# B&R Automation Studio project AriesV2
Automation Studio 4.2.4.149

## Configuration Config_3500HS

### Task classes (Cpu.sw)
```
Cyclic#1:
  runFirst <- Libraries.wbrServices.InitSP.runFirst.prg (BuildOptions=-D "str(x)=#x" -D AS_PROJ=str($(AS_PROJECT_NAME)) -D AS_CFG=str($(AS_CONFIGURATION)) -D "AS_VERS=str($(AS_VERSION))" -D "AS_USER=str($(AS_USER_NAME))" -D "AS_CMPNY=str($(AS_COMPANY_NAME))")
  ForceIO1 <- HMI.ForceIO.prg
  ForceIO <- HMI.ForceIO.prg
Cyclic#8:
  wbrService <- Libraries.wbrServices.Cyclic.wbrService.prg
  HMITableMa <- HMI.HMITableManager.prg
  Recipe_Han <- Auxiliary_Services_Control.Recipe_Handling.prg  // Call functions that manage structures pertaining to params
  hmilogic <- HMI.hmilogic.prg
  ComLogger <- Auxiliary_Services_Control.ComLogger.prg [disabled]
  File_Handl <- Auxiliary_Services_Control.File_Handling.prg
DataObjects: ethIPcon
VcDataObjects: VisuW1 <- HMI.VisuW1.dob
Binaries: TCData, vccpwd, vccbtn, vcpdvnc, arialbd, vcmgr, vctcal, vcfile, vccnum, vcfntttf, vcgclass, vcbclass, vccshape, vccstr, vccalarm, vccscale, arial, vcalarm, vcdsloc, vcchtml, vccdt, vccbmp, vcshared, vcxml, vccurl, vcrt, vcctext, vcnet, vcclbox, vcdsint, vcpdsw, vccovl, vccline, VisuW101, VisuW102, VisuW103, vera, vccgauge, vcpfx20, TC, Data_Log, MAPP_Alm, MAPP_Rec, MAPP_Web, MAPP_File, MAPP_Cfg, iomap, asfw, sysconf, ashwd, arconfig, Alarm, vcctrend, vccpopup, vccddbox, vccpiech, vcpkat, verabd, Visu, Visu02, Visu03, Visu01, Axes, Config_1, MAPP_Com, Recipe, File_Mgmt, vccslider, Acp10Map1, User, Role, Data, Config, VisuW03, VisuW02, VisuW01, acp10cfg, Acp10map, Acp10sys, vcpfar00
Libraries: wbrsprintf, FileIO, AsXml, standard, runtime, astime, brsystem, sys_lib, AsANSL, AsARCfg, AsBrMath, AsBrStr, DataObj, AsTCP, AsUDP, AsUSB, MpCom, MpAlarm, MpFile, MpRecipe, MpWebXs, AsArSdm, AsIecCon, operator, AsIOTime, AsMem, AsArLog, AsArProf, MTBasics, MTTypes, MTFilter, jgLibC, MTData, ArTextSys, AsICMP, bglibasWBR, MAPPSuppor, wbrFltUtil, wbrListSvc, wbrLogSvc, wbrMemSvc, wbrPingSvc, vcresman, arsvcreg, ashw, AsMbTCP, AsSafety, powerlnk
```

### MAPP_Cfg.mprecipecsv - X20CP1301/mapp/MAPP_Cfg.mprecipecsv
```
Element Config_CSV_MpLink (Type=mprecipecsv)
  mapp.Recipe.Csv:
    Format:
      DecimalMark = .
```

## Configuration Config_Deployment

### Task classes (Cpu.sw)
```
Cyclic#1 (cycle 4000 us, tolerance 0 us):
  ForceIO <- HMI.ForceIO.prg
  Creaser <- Application.Creaser.prg
  ForceIO1 <- HMI.ForceIO.prg
Cyclic#8 (cycle 8000 us, tolerance 30000000 us):
  LineContro <- MotionControl.LineControl.prg
  Recipe_Han <- Auxiliary_Services_Control.Recipe_Handling.prg
  hmilogic <- HMI.hmilogic.prg
  HMITableMa <- HMI.HMITableManager.prg
  File_Handl <- Auxiliary_Services_Control.File_Handling.prg
  ComLogger <- Auxiliary_Services_Control.ComLogger.prg
DataObjects: ethIPcon
NcDataObjects: acp10etxen <- acp10etxen.dob, Axisa <- Axisobj.Axisa.dob, Axisi <- Axisobj.Axisi.dob
VcDataObjects: Visu1 <- HMI.Visu.dob
Binaries: vccpwd, vccbtn, arialbd, vcfile, vccnum, vcfntttf, vcgclass, vcbclass, vccshape, vccstr, vccalarm, vccscale, arial, vcalarm, vcdsloc, vcchtml, vccdt, vccbmp, vcshared, vcxml, vccurl, vcrt, vcctext, vcclbox, vcdsint, vcpdsw, vccovl, vccline, vera, vcpfar00, vcpkat, vccddbox, vccpopup, vcnet, vctcal, vcmgr, vcpdvnc, udbdef, Acp10sys, TCData, Visu102, Visu101, Visu103, Alarm, ashwd, asfw, MAPP_Cfg, MAPP_File, MAPP_Web, MAPP_Rec, MAPP_Alm, Data_Log, arconfig, sysconf, iomap, Config, acp10cfg, Acp10map, VisuW101, vcpfx20, vcctrend, vccpiech, verabd, Visu, Visu02, Visu03, Visu01, Axes, Config_1, MAPP_Com, Recipe, File_Mgmt, vccslider, Acp10Map1, User, Role, Data, VisuW03, VisuW02, VisuW01, TC, vccgauge, VisuW103, VisuW102
Libraries: FileIO, AsXml, standard, runtime, astime, brsystem, sys_lib, AsANSL, AsARCfg, AsBrMath, AsBrStr, DataObj, AsTCP, AsUDP, AsUSB, AsArSdm, AsIecCon, operator, AsIOTime, AsMem, AsArLog, AsArProf, AsICMP, Acp10man, Acp10par, NcGlobal, Acp10_MC, MpAxis, MpCom, wbrsprintf, wbrPingSvc, wbrMemSvc, wbrLogSvc, wbrListSvc, wbrFltUtil, MpWebXs, MpRecipe, MpFile, MpAlarm, MAPPSuppor, jgLibC, bglibasWBR, vcresman, arsvcreg, powerlnk, Acp10sim, ashw, AsMbTCP, AsSafety, ArTextSys
```

### Hardware
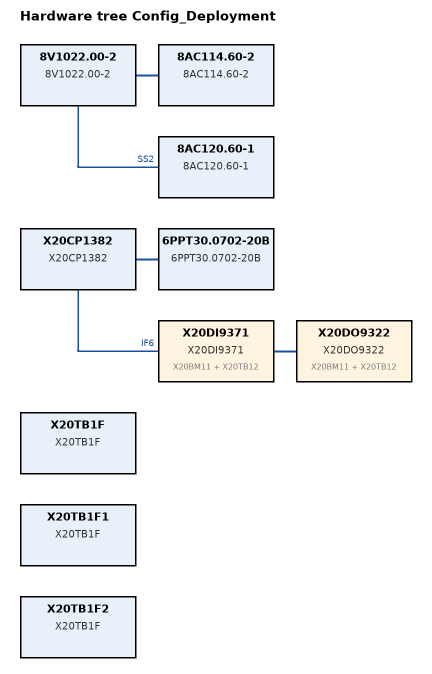
```
6PPT30.0702-20B : 6PPT30.0702-20B v1.1.0.0  [ETH1 -> X20CP1382.IF2 (NodeNumber=1)]
  Terminal = true
  Startmode = 1
  ShowBootlogoVNC = 1
  Mode = Manual
  InternetAddress = 192.168.10.20
  DefaultGateway = 192.168.10.1
  Subnetmask = 255.255.255.0
  Displaybrightness = 75
  SelectedFavoriteVNC = 192.168.10.10
  Favorites_VNC1 = 192.168.10.10
  PasswordVNC = 
  PasswordCIFS = 
  PasswordService = 
  PPTImage = PPT_30_V1.1.1
  VncRefreshRate = 200
8AC114.60-2 : 8AC114.60-2 v1.0.0.8  [SS -> 8V1022.00-2.SS1; PLK1 -> X20CP1382.IF3 (NodeNumber=2)]
8AC120.60-1 : 8AC120.60-1 v1.0.0.2  [SS -> 8V1022.00-2.SS2]
8V1022.00-2 : 8V1022.00-2 v1.0.0.2
  AxisIsPeriodic_r1 = on
  BothEndSwitchesAreNormallyOpen_r1 = on
  QuickStopIsNormallyOpen_r1 = on
X20BM11 : X20BM11 v1.0.0.1  [X2X1 -> X20CP1382.IF6]
X20BM11a : X20BM11 v1.0.0.1  [X2X1 -> X20BM11.X2X2]
X20CP1382 : X20CP1382 v1.3.0.0  [X1 -> X1.SL; X2 -> X2.SL; X3 -> X3.SL]
  Module X1 (Type=X1, Virtual=true, Version=1.0.0.0)
    Connection (Connector=SS1, TargetModule=X20TB1F, TargetConnector=SS)
    Connection (Connector=SL, TargetModule=X20CP1382, TargetConnector=X1)
  Module X2 (Type=X2, Virtual=true, Version=1.0.0.0)
    Connection (Connector=SS1, TargetModule=X20TB1F1, TargetConnector=SS)
    Connection (Connector=SL, TargetModule=X20CP1382, TargetConnector=X2)
  Module X3 (Type=X3, Virtual=true, Version=1.0.0.0)
    Connection (Connector=SS1, TargetModule=X20TB1F2, TargetConnector=SS)
    Connection (Connector=SL, TargetModule=X20CP1382, TargetConnector=X3)
  Connector IF2:
    ActivateDevice = 1
    HostName = x20cpu
    Mode = Manual
    InternetAddress = 192.168.10.10
    SubnetMask = 255.255.255.0
    InaNodeNumber = 0
    Vnc1
    VncVcObjectName1 = Visup
    VncKeyMappingFile1 = VC\PS2-Keyboard4.dis
    VncRefreshRate1 = 200
  Connector IF3:
    CycleTime = 4000
  Connector IF6:
    CycleTime = 4000
  ConfigurationID = AriesV2_Config_Test
  UserPartitionSize = 256
  UserRamSize = 5000
  RemMemSize = 25000
  PermanentPvSize = 15000
  VolatileGlobalPvSize = 300000
  RebootReset = 2
  RebootPowerfail = 2
  TimerDeviceType = EPLX2X
  TimerDevice = X20CP1382.IF3
  TaskClassIdleTime = 8000
  Cyclic1Duration = 4000
  Cyclic1Tolerance = 0
  Cyclic2Duration = 16000
  Cyclic2Tolerance = 16000
  Cyclic3Duration = 48000
  Cyclic3Tolerance = 48000
  Cyclic4Duration = 96000
  Cyclic4Tolerance = 96000
  Cyclic5Duration = 200000
  Cyclic5Tolerance = 200000
  Cyclic6Duration = 496000
  Cyclic6Tolerance = 496000
  Cyclic7Duration = 1000000
  Cyclic7Tolerance = 1000000
  Cyclic8Duration = 8000
  Cyclic8Tolerance = 30000000
  FileDevice1
  FileDeviceName1 = ROOT
  FileDevicePath1 = F:\
  FileDevice2
  FileDeviceName2 = Config
  FileDevicePath2 = F:\Config
  FileDevice3
  FileDeviceName3 = Recipe
  FileDevicePath3 = F:\Recipe
  FileDevice4
  FileDeviceName4 = Process
  FileDevicePath4 = F:\Process
  FtpUser1
  FtpUsername1 = admin
  FtpUserPassword1 = tXcQUdKIsoY/H/jtKSqzHLRzyWbO/eZFb+QmJVs8vuM=
  FtpUserSalt1 = fFlgpUU6
  FTPAccessRight1 = 0
  FTPdevice1 = ALL
  FtpUser2
  FtpUsername2 = user
  FtpUserPassword2 = M/sBBWLbPcMSL0ECBo9+NNWk5QFExAfaSSh+paOlJpQ=
  FtpUserSalt2 = diDYFxUT
  FTPAccessRight2 = 0
  FTPMSpath2 = /
X20DI9371 : X20DI9371 v1.0.1.3  [SS1 -> X20TB12.SS; SL -> X20BM11.SL1]
  Supervision = off
X20DO9322 : X20DO9322 v1.0.3.0  [SS1 -> X20TB12a.SS; SL -> X20BM11a.SL1]
  Supervision = off
X20TB12 : X20TB12 v1.0.0.0
X20TB12a : X20TB12 v1.0.0.0
X20TB1F : X20TB1F v1.0.0.0
X20TB1F1 : X20TB1F v1.0.0.0
X20TB1F2 : X20TB1F v1.0.0.0
```

### Acp10cfg.ncc - X20CP1382/Motion/Acp10cfg.ncc
```
NcConfiguration (Version=3.16.1, NcSwId=Acp10)
  ACP10CF1_typ:
    cnt_nettrc_rec_drive = 1500
    bufsize_trace_upload = 1200
    tc_nc_man_task = Cyclic #1
    glob_pv_as_ncobject = Yes
    ncsys_dl_broadcast = Yes
    ncsys_dl_acp_reset = Yes
    safemc_log_err_to_ax = Yes
    network_init:
      ncsw_init_execute = Yes
      automatic_execute = Yes
      node_nr_warning = Yes
      net_err_before_ncact = Yes
    nettrc:
      enter_parsecrec = Yes
      enter_ncaction = Yes
      save_ring_startidx = Yes
    cam_prof_download:
      cam_dat_dl_parallel = No
      tc_cam_dl_parallel = Task class for NC Manager task
    plk_if[0]:
      if_name = IF3
      tc_CycDat_PLCopen = Task class for NC Manager task
      mc_broadcast_extdat = No
```

### MAPP_File.mpfilemanagerui - X20CP1382/mapp/MAPP_File.mpfilemanagerui
```
Element File_Manager_MpLink (Type=mpfilemanagerui)
```

## Configuration Config_Test

CPU X20CP1584, AutomationRuntime B4.26, Build 4.1.2, Vc V4.26.3, Safety 0.0

CPU X20CP1585, AutomationRuntime B4.26, Build 4.1.2, Vc V4.26.3, Safety 1.5

### Task classes (Cpu.sw)
```
Cyclic#1 (cycle 8000 us, tolerance 0 us):
  ForceIO <- HMI.ForceIO.prg
  Creaser <- Application.Creaser.prg
  ForceIO1 <- HMI.ForceIO.prg
Cyclic#8 (cycle 8000 us, tolerance 30000000 us):
  LineContro <- MotionControl.LineControl.prg
  Recipe_Han <- Auxiliary_Services_Control.Recipe_Handling.prg
  hmilogic <- HMI.hmilogic.prg
  HMITableMa <- HMI.HMITableManager.prg
  File_Handl <- Auxiliary_Services_Control.File_Handling.prg
  ComLogger <- Auxiliary_Services_Control.ComLogger.prg
DataObjects: ethIPcon
NcDataObjects: acp10etxen <- acp10etxen.dob, Axisa <- Axisobj.Axisa.dob, Axisi <- Axisobj.Axisi.dob
VcDataObjects: Visu1 <- HMI.Visu.dob
Binaries: vccpwd, vccbtn, arialbd, vcfile, vccnum, vcfntttf, vcgclass, vcbclass, vccshape, vccstr, vccalarm, vccscale, arial, vcalarm, vcdsloc, vcchtml, vccdt, vccbmp, vcshared, vcxml, vccurl, vcrt, vcctext, vcclbox, vcdsint, vcpdsw, vccovl, vccline, VisuW102, VisuW103, vera, vccgauge, TC, vcpfar00, VisuW01, VisuW02, VisuW03, Data, Role, User, Acp10Map1, vccslider, File_Mgmt, Recipe, MAPP_Com, Config_1, Axes, Visu01, Visu03, Visu02, Visu, verabd, vcpkat, vccpiech, vccddbox, vccpopup, vcctrend, vcpfx20, VisuW101, vcnet, vctcal, vcmgr, vcpdvnc, Acp10map, acp10cfg, Config, iomap, sysconf, arconfig, Data_Log, MAPP_Alm, MAPP_Rec, MAPP_Web, MAPP_File, MAPP_Cfg, asfw, ashwd, Alarm, udbdef, Acp10sys, TCData
Libraries: FileIO, AsXml, standard, runtime, astime, brsystem, sys_lib, AsANSL, AsARCfg, AsBrMath, AsBrStr, DataObj, AsTCP, AsUDP, AsUSB, AsArSdm, AsIecCon, operator, AsIOTime, AsMem, AsArLog, AsArProf, AsICMP, Acp10man, Acp10par, NcGlobal, Acp10_MC, MpAxis, MpCom, wbrsprintf, wbrPingSvc, wbrMemSvc, wbrLogSvc, wbrListSvc, wbrFltUtil, MpWebXs, MpRecipe, MpFile, MpAlarm, MAPPSuppor, jgLibC, bglibasWBR, vcresman, AsSafety, AsMbTCP, ashw, arsvcreg, powerlnk, Acp10sim
```

### Task classes (Cpu.sw)
```
Cyclic#1 (cycle 8000 us, tolerance 0 us):
  ForceIO <- HMI.ForceIO.prg
  Creaser <- Application.Creaser.prg
  ForceIO1 <- HMI.ForceIO.prg
DataObjects: ethIPcon
NcDataObjects: acp10etxen <- acp10etxen.dob, Axisa <- Axisobj.Axisa.dob, Axisi <- Axisobj.Axisi.dob
Binaries: TCData, Acp10sys, udbdef, Acp10map, acp10cfg, Config, iomap, sysconf, arconfig, Data_Log, MAPP_Alm, MAPP_Rec, MAPP_Web, MAPP_File, MAPP_Cfg, asfw, ashwd, Alarm, vccpwd, vccbtn, arialbd, vcfile, vccnum, vcfntttf, vcgclass, vcbclass, vccshape, vccstr, vccalarm, vccscale, arial, vcalarm, vcdsloc, vcchtml, vccdt, vccbmp, vcshared, vcxml, vccurl, vcrt, vcctext, vcclbox, vcdsint, vcpdsw, vccovl, vccline, VisuW102, VisuW103, vera, vccgauge, TC, vcpfar00, VisuW01, VisuW02, VisuW03, Data, Role, User, Acp10Map1, vccslider, File_Mgmt, Recipe, MAPP_Com, Config_1, Axes, Visu01, Visu03, Visu02, Visu, verabd, vcpkat, vccpiech, vccddbox, vccpopup, vcctrend, vcpfx20, VisuW101, vcnet, vctcal, vcmgr, vcpdvnc
Libraries: FileIO, AsXml, standard, runtime, astime, brsystem, sys_lib, AsANSL, AsARCfg, AsBrMath, AsBrStr, DataObj, AsTCP, AsUDP, AsUSB, AsArSdm, AsIecCon, operator, AsIOTime, AsMem, AsArLog, AsArProf, AsICMP, powerlnk, Acp10man, Acp10par, NcGlobal, Acp10_MC, MTBasics, MTTypes, MpAxis, MpCom, wbrsprintf, wbrPingSvc, wbrMemSvc, wbrLogSvc, wbrListSvc, wbrFltUtil, MTProfile, MTFilter, MTData, MpWebXs, MpRecipe, MpFile, MpAlarm, MAPPSuppor, jgLibC, bglibasWBR, ArTextSys, vcresman, AsSafety, AsMbTCP, ashw, arsvcreg
```

### Task classes (Cpu.sw)
```
Cyclic#1 (cycle 8000 us, tolerance 0 us):
  runFirst <- Libraries.wbrServices.InitSP.runFirst.prg (BuildOptions=-D "str(x)=#x" -D AS_PROJ=str($(AS_PROJECT_NAME)) -D AS_CFG=str($(AS_CONFIGURATION)) -D "AS_VERS=str($(AS_VERSION))" -D "AS_USER=str($(AS_USER_NAME))" -D "AS_CMPNY=str($(AS_COMPANY_NAME))")
  ForceIO1 <- HMI.ForceIO.prg
  ForceIO <- HMI.ForceIO.prg
Cyclic#8 (cycle 8000 us, tolerance 30000000 us):
  wbrService <- Libraries.wbrServices.Cyclic.wbrService.prg
  HMITableMa <- HMI.HMITableManager.prg
  Recipe_Han <- Auxiliary_Services_Control.Recipe_Handling.prg  // Call functions that manage structures pertaining to params
  hmilogic <- HMI.hmilogic.prg
  ComLogger <- Auxiliary_Services_Control.ComLogger.prg
  File_Handl <- Auxiliary_Services_Control.File_Handling.prg
DataObjects: ethIPcon
Binaries: vccpwd, vccbtn, arialbd, vcfile, vccnum, vcfntttf, vcgclass, vcbclass, vccshape, vccstr, vccalarm, vccscale, arial, vcalarm, vcdsloc, vcchtml, vccdt, vccbmp, vcshared, vcxml, vccurl, vcrt, vcctext, vcclbox, vcdsint, vcpdsw, vccovl, vccline, VisuW102, VisuW103, vera, vccgauge, Alarm, ashwd, asfw, MAPP_Cfg, MAPP_File, MAPP_Web, MAPP_Rec, MAPP_Alm, Data_Log, TC, vcpfar00, Acp10sys, Acp10map, acp10cfg, VisuW01, VisuW02, VisuW03, Config, Data, Role, User, Acp10Map1, vccslider, File_Mgmt, Recipe, MAPP_Com, Config_1, Axes, Visu01, Visu03, Visu02, Visu, verabd, vcpkat, vccpiech, vccddbox, vccpopup, vcctrend, arconfig, sysconf, iomap, vcpfx20, VisuW101, vcnet, vctcal, vcmgr, vcpdvnc, TCData
Libraries: wbrsprintf, FileIO, AsXml, standard, runtime, astime, brsystem, sys_lib, AsANSL, AsARCfg, AsBrMath, AsBrStr, DataObj, AsTCP, AsUDP, AsUSB, MpCom, MpAlarm, MpFile, MpRecipe, MpWebXs, AsArSdm, AsIecCon, operator, AsIOTime, AsMem, AsArLog, AsArProf, MTBasics, MTTypes, MTFilter, jgLibC, MTData, ArTextSys, AsICMP, bglibasWBR, MAPPSuppor, wbrFltUtil, wbrListSvc, wbrLogSvc, wbrMemSvc, wbrPingSvc, vcresman, arsvcreg, powerlnk, AsSafety, AsMbTCP, ashw
```

### Hardware
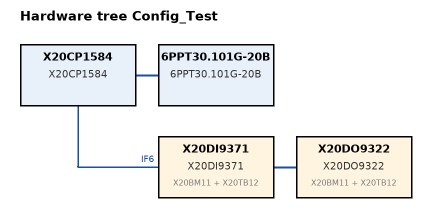
```
6PPT30.101G-20B : 6PPT30.101G-20B v1.1.0.0  [ETH1 -> X20CP1584.IF2 (NodeNumber=1)]
  Terminal = true
  PasswordVNC = 
  PasswordCIFS = 
  PasswordService = 
  VncKeyMappingFile = VC\6PPT30.101G-20B.dis
  VncPortNumber = 5901
X20BM11 : X20BM11 v1.0.0.1  [X2X1 -> X20CP1584.IF6]
X20BM11a : X20BM11 v1.0.0.1  [X2X1 -> X20BM11.X2X2]
X20CP1584 : X20CP1584 v1.3.2.0
  Connector IF2:
    ActivateDevice = 1
    EthInterfaceRedundant = 0
    HostName = x20cpu
    Mode = Manual
    InternetAddress = 192.168.10.10
    SubnetMask = 255.255.255.0
    Vnc1
    VncVcObjectName1 = Visu1
    VncKeyMappingFile1 = VC\PS2-Keyboard4.dis
    VncRefreshRate1 = 200
  Connector IF3:
    EplInterfaceRedundant = 0
    CycleTime = 8000
    EplEthInterfaceRedundant = 0
  Connector IF6:
    CycleTime = 8000
  ConfigurationID = AriesV2_Config_Test
  UserRamSize = 5000
  RemMemSize = 25000
  PermanentPvSize = 15000
  VolatileGlobalPvSize = 300000
  RebootReset = 2
  RebootPowerfail = 2
  TimerDeviceType = EPLX2X
  TimerDevice = X20CP1584.IF3
  TaskClassIdleTime = 8000
  Cyclic1Duration = 8000
  Cyclic1Tolerance = 0
  Cyclic2Duration = 16000
  Cyclic2Tolerance = 16000
  Cyclic3Duration = 48000
  Cyclic3Tolerance = 48000
  Cyclic4Duration = 96000
  Cyclic4Tolerance = 96000
  Cyclic5Duration = 200000
  Cyclic5Tolerance = 200000
  Cyclic6Duration = 496000
  Cyclic6Tolerance = 496000
  Cyclic7Duration = 1000000
  Cyclic7Tolerance = 1000000
  Cyclic8Duration = 8000
  Cyclic8Tolerance = 30000000
  FileDevice1
  FileDeviceName1 = ROOT
  FileDevicePath1 = F:\
  FileDevice2
  FileDeviceName2 = Config
  FileDevicePath2 = F:\Config
  FileDevice3
  FileDeviceName3 = Recipe
  FileDevicePath3 = F:\Recipe
  FileDevice4
  FileDeviceName4 = Process
  FileDevicePath4 = F:\Process
X20DI9371 : X20DI9371 v1.0.2.0  [SS1 -> X20TB12.SS; SL -> X20BM11.SL1]
  Supervision = off
X20DO9322 : X20DO9322 v1.0.3.0  [SS1 -> X20TB12a.SS; SL -> X20BM11a.SL1]
  Supervision = off
X20TB12 : X20TB12 v1.0.0.0
X20TB12a : X20TB12 v1.0.0.0
```

### Acp10map.ncm - X20CP1382/Motion/Acp10map.ncm
```
NcMapping (NcSwId=Acp10, DisabledNodesAreHidden=False)
  NcObject Axis1 (ModuleId=8V1022.00-2, Type=ncAXIS, Channel=1, AcoposSimulation=Complete, InitParameter=Axisi, AcoposParameter=Axisa, AdditionalData=PLCopen_ModPos="1000,1" , Disabled=FALSE, ModuleDisabled=FALSE)
  NcObject 8V1045.00-2_ncV_AXIS1 (ModuleId=8V1022.00-2, Type=ncV_AXIS, Channel=1, Disabled=TRUE, ModuleDisabled=FALSE)
```

### MAPP_Web.mpwebxs - X20CP1382/mapp/MAPP_Web.mpwebxs
```
Element WebXs (Type=mpwebxs)
```

### IoMap.iom - X20CP1584/IoMap.iom
```iecst
VAR_CONFIG
	IO.iSafeMachineState AT %IX."X20DI9371".DigitalInput01;
	IO.iCreaserShaftSensor AT %IX."X20DI9371".DigitalInput02;
	IO.iFiberOpticSensor AT %IX."X20DI9371".DigitalInput03;
	IO.iSM1Disabled AT %IX."X20DI9371".DigitalInput05;
	IO.oBoardFeedingLight  AT %QX."X20DO9322".DigitalOutput05;
	IO.oCreaserCCWRotation   AT %QX."X20DO9322".DigitalOutput03;
	IO.oCreaserCWRotation   AT %QX."X20DO9322".DigitalOutput04;
	IO.oUIIndicatorLight  AT %QX."X20DO9322".DigitalOutput07;
END_VAR
```

### Acp10cfg.ncc - X20CP1584/Motion/Acp10cfg.ncc
```
NcConfiguration (Version=3.16.0, NcSwId=Acp10)
  ACP10CF1_typ:
    cnt_nettrc_rec_drive = 1500
    bufsize_trace_upload = 1200
    tc_nc_man_task = Cyclic #1
    glob_pv_as_ncobject = Yes
    ncsys_dl_broadcast = Yes
    ncsys_dl_acp_reset = Yes
    safemc_log_err_to_ax = Yes
    network_init:
      ncsw_init_execute = Yes
      automatic_execute = No
      node_nr_warning = Yes
      net_err_before_ncact = Yes
    nettrc:
      enter_parsecrec = Yes
      enter_ncaction = Yes
      save_ring_startidx = Yes
    cam_prof_download:
      cam_dat_dl_parallel = No
      tc_cam_dl_parallel = Task class for NC Manager task
    plk_if[0]:
      if_name = IF3
      tc_CycDat_PLCopen = Task class for NC Manager task
      mc_broadcast_extdat = No
```

### MAPP_Rec.mprecipecsv - X20CP1584/mapp/MAPP_Rec.mprecipecsv
```
Element Recipe_CSV_MpLink (Type=mprecipecsv)
  mapp.Recipe.Csv:
    Format:
      DecimalMark = .
```

## Logical view

Binary libraries used (declarations not repeated): operator, runtime, astime, AsIecCon, FileIO, AsXml, standard, brsystem, sys_lib, AsANSL, AsARCfg, AsBrMath, AsBrStr, DataObj, AsTCP, AsUDP, AsUSB, AsArSdm, AsIOTime, AsMem, AsArLog, AsArProf, MTTypes, jgLibC, MAPPSuppor, wbrsprintf, wbrListSvc, wbrPingSvc, AsICMP, MpCom, MpAxis 1.60.1, MpWebXs 1.20.5, MpRecipe 1.20.5, MpAlarm, MpFile, ArTextSys, Acp10man, Acp10par 3.16.2, NcGlobal, Acp10sim 3.16.1, Acp10_MC, MTData, MTBasics 2.21.0, MTFilter 2.10.0

### GlobalConstants.var
```iecst
VAR CONSTANT
	FORCEIO_ACCESS_LEVEL : UINT := 1;
	CONFIG_ACCESS_LEVEL : UINT := 2;
	RECIPE_ACCESS_LEVEL : UINT := 1;
	DEFINE_MENU_L_HIDE_TIMEOUT_MS : UDINT := 7000;
	DEFINE_MENU_R_HIDE_TIMEOUT_MS : UDINT := 7000;
	DEFINE_HMI_SPLASHSCREEN_TO_MS : UDINT := 5000;
	MAX_IDX_TOTAL_RECIPES : UINT := 100;
	DEFINE_LOGIN_TO : REAL := 600; (*// at timer DEFINE_LOGIN_TO * 1000 *60*)
END_VAR
(*Insert your comment here.*)
VAR CONSTANT
	MAX_IDX_CREASES : UDINT := 9;
END_VAR
```

### Machine.typ
```iecst
TYPE
	CreaserPrcsState_Enum :
		( (*Make sure the indices entered below line up with the VC texts displayed on the UI*)
		PRCS_STATE_INIT := 0,
		PRCS_STATE_READY := 1,
		PRCS_STATE_FEED_BOARD := 2,
		PRCS_STATE_MOVE_CREASE := 3,
		PRCS_STATE_CREASE := 4,
		PRCS_STATE_MOVE_CREASE_WIDTH := 5,
		PRCS_STATE_ERROR := 6,
		PRCS_STATE_EJECT_FINISHED_BOARD := 7,
		PRCS_STATE_SOFT_STOP := 8,
		PRCS_STATE_MOVE_PHOTOEYE_OFFSET := 9
		);
	AriesMachineState_Enum :
		( (*Make sure the indices entered below line up with the VC texts displayed on the UI*)
		MACHINE_STATE_INIT := 0,
		MACHINE_STATE_IDLE := 1,
		MACHINE_STATE_RUNNING := 2,
		MACHINE_STATE_ERROR := 3,
		MACHINE_STATE_HARDWARE_INIT := 4,
		MACHINE_STATE_AXIS_POWER := 5,
		MACHINE_STATE_AXIS_HOME := 6,
		MACHINE_STATE_MANUAL_EJECT := 7
		);
END_TYPE

(*Insert your comment here.*)

TYPE
	CreaserConfig_typ : 	STRUCT
		FeedAxisAccel : REAL;
		FeedAxisDecel : REAL;
		PhotoEyeOffset : REAL;
		PreInsertSpeed : REAL;
		BoardLengthTolerance : REAL;
		CreaseInfeedDelay : REAL;
		BypassBoardLengthError : UDINT;
	END_STRUCT;
	AriesCreaserParams_typ : 	STRUCT
		CreaseDistance_mm : ARRAY[0..MAX_IDX_CREASES]OF REAL;
		CreaseWidth_mm : REAL;
		CreaseCount : UDINT;
		ShaftSensorEdge : UDINT;
		CreaserDirection : UDINT;
		CreaserMotorIdxLag_S : REAL;
		TotalBoardLength : REAL;
	END_STRUCT;
END_TYPE

(*Insert your comment here.*)

TYPE
	AriesIOPoints_typ : 	STRUCT
		oCreaserCCWRotation : BOOL;
		oCreaserCWRotation : BOOL;
		oBoardFeedingLight : BOOL;
		oUIIndicatorLight : BOOL;
		iSafeMachineState : BOOL;
		iCreaserShaftSensor : BOOL;
		iFiberOpticSensor : BOOL;
		iSM1Disabled : BOOL;
	END_STRUCT;
END_TYPE

(*Insert your comment here.*)

TYPE
	Machine_Alarms_typ : 	STRUCT  (*Did something fancy here- structure is copied into array for VC error texts, make sure the following numbers line up with the VC error text indices!*)
		SM1_Disabled : BOOL; (*0*)
		Unsafe_Machine_State : BOOL; (*1*)
		Fiber_Optic_Blocked_RunCmd : BOOL; (*2*)
		Creaser_Shaft_Edge_Timeout : BOOL; (*3*)
		Error_State_Unsafe_Machine : BOOL; (*4*)
		Error_State_SM1_Power : BOOL; (*5*)
		Feed_Axis_Motor_Error : BOOL; (*6*)
		Crease_Count_Greater_Max : BOOL; (*7*)
		Error_State_Process_Error : BOOL; (*8*)
		Load_Recipe : BOOL; (*9*)
		Manual_Home_Creaser_Blade : BOOL; (*10*)
		Board_Length_GT_Confgd_Amount : BOOL; (*11*)
		Board_Length_LT_Confgd_Amount : BOOL; (*12*)
		Measured_Length_GT_Configured : BOOL; (*13*)
		Measured_Length_LT_Configured : BOOL; (*14*)
		Unsaved_Recipe_Params : BOOL; (*15*)
	END_STRUCT;
	Global_Statistics_typ : 	STRUCT
		total_runtime : UDINT;
		runtime_h : UDINT;
		runtime_m : UDINT;
		runtime_s : UDINT;
		total_processed : UDINT;
		Reset : BOOL;
		total_creases : UDINT;
		Sum_Board_Travel_Lengths : REAL;
		Avg_Board_Length : REAL;
	END_STRUCT;
END_TYPE
```

### Generic_Rec_Cfg.typ
```iecst
TYPE
	HMIConfig_typ : 	STRUCT
		passwordSetup : STRING[15];
		passwordEngineer : STRING[15];
		passwordFactory : STRING[15];
		MachineLang : UDINT;
	END_STRUCT;
END_TYPE

(*Insert your comment here.*)

TYPE
	Global_Rec_typ : 	STRUCT
		MagicPrefix : UDINT;
		FeedVelocity : REAL;
		Crease : AriesCreaserParams_typ;
		MagicSuffix : UDINT;
	END_STRUCT;
	Global_Cfg_typ : 	STRUCT
		MagicPrefix : UDINT;
		Creaser : CreaserConfig_typ;
		HMI : HMIConfig_typ;
		wbrMemService : wbrMemService_typ;
		cfgCompile : cfgCompileVersionInfo_typ;
		MagicSuffix : UDINT;
	END_STRUCT;
END_TYPE

(*Insert your comment here.*)

TYPE
	Global_Rec_Cfg_typ : 	STRUCT
		Rec : Global_Rec_typ;
		Cfg : Global_Cfg_typ;
	END_STRUCT;
	Global_RecCfg_Public_In_typ : 	STRUCT
		Copy_default_to_save : USINT;
		Copy_default_to_active : USINT;
		Copy_save_to_active : USINT;
		Copy_save_to_default : USINT;
		Copy_active_to_save : USINT;
		Copy_active_to_default : USINT;
		Copy_internal_to_default : USINT;
		FileName : STRING[255];
	END_STRUCT;
	Global_RecCfg_Public_Out_typ : 	STRUCT
		save_differs_from_active : USINT;
		default_differs_from_save : USINT;
		active_differs_from_default : USINT;
	END_STRUCT;
	Global_Rec_Cfg_Info_typ : 	STRUCT
		O : Global_RecCfg_Public_Out_typ;
		I : Global_RecCfg_Public_In_typ;
	END_STRUCT;
	Global_Rec_Cfg_IO_typ : 	STRUCT
		Rec : Global_Rec_Cfg_Info_typ;
		Cfg : Global_Rec_Cfg_Info_typ;
	END_STRUCT;
	Global_Par_typ : 	STRUCT
		save : Global_Rec_Cfg_typ;
		active : Global_Rec_Cfg_typ;
		defaultvals : Global_Rec_Cfg_typ;
		IO : Global_Rec_Cfg_IO_typ;
	END_STRUCT;
END_TYPE

(*Insert your comment here.*)
```

### Package Logical/Libraries - Global libraries

### Package Logical/Libraries/wbrServices - Service libraries

### Library Logical/Libraries/wbrServices/wbrMemSvc (ANSIC) - Allocate heap memory using AsMem

#### wbrMemSvc.c
```c
/********************************************************************
 * \copyright -- Piedmont Automation
 ********************************************************************
 * Program : wbrMemSvc
 * \file :   wbrMemSvc.c
 * \author : Blanton Radford
 * \date Created: April 14, 2016
 ******************************************************************* /
 * Implementation of library wbrListSvc
 ********************************************************************/

#include "wbrMemSvc.h"

AsMemPartAllocClear_typ   allocate;
AsMemPartFree_typ         freeMem;
AsMemPartRealloc_typ      reAllocate;
AsMemPartInfo_typ         memInfo;

/*! \todo
*/
UDINT memSvcAllocate(UDINT size)
{
  allocate.len=     size;
  AsMemPartAllocClear(&allocate);
  if(allocate.status == 0)  return  allocate.mem;

  //! \todo   handle errors
  return  0;
}

/*! \brief Init-SP for AsMem heap memory and linked list services
    \warning   this init must be called in the first Init-SP in TC#1
*/
BOOL initMemSvc(UDINT partitionSize)
{
 AsMemPartCreate_typ  getMem;

  getMem.enable=
      allocate.enable=
      freeMem.enable=
      reAllocate.enable=
      memInfo.enable=         1;

  getMem.len=     partitionSize;

  AsMemPartCreate(&getMem);

  allocate.ident=
      freeMem.ident=
      reAllocate.ident=
      memInfo.ident=          getMem.ident;

  return  (BOOL)allocate.ident;
}

/*! \brief    Frees a block of heap memory

    \pre      \todo
    \warning  \todo

*/
UINT  memSvcFree(UDINT block)
{
  if(!block)
  {
    //! \todo   report null address
    return  0xAAAA;
  }

  freeMem.mem=  block;
  AsMemPartFree(&freeMem);

  if(freeMem.status != 0)
  {
    //!   \todo   possibly loop to try again n times?
    //!   \todo   handle error, flag address for later memory cleanup
  }

  return  freeMem.status;
}

/*! \brief    Returns size of the largest available memory block

    \pre      \todo
    \warning  \todo
    \todo

**/
UDINT memSvcGetMemInfo()
{
  AsMemPartInfo(&memInfo);

  return   memInfo.maxBlockSizeFree;
}
```

### Library Logical/Libraries/wbrServices/wbrLogSvc (ANSIC) - Logging to logbooks, other logs todo
Depends on: AsArLog, wbrListSvc, wbrsprintf

### Library Logical/Libraries/wbrServices/bglibasWBR (ANSIC) - Modified by WBR beginning 2015-01-13

#### bglibasWBR.fun
```iecst
(********************************************************************
 * COPYRIGHT -- belgor
 ********************************************************************
 * Library: bglibas
 * File: bglibas.fun
 * Author: admin
 * Created: March 07, 2012
 ********************************************************************
 * Functions and function blocks of library bglibas
 ********************************************************************)
(*=========================================================================*)
(*SUPPORT FOR SIMPLE STATE MACHINE (SSM)*)
(*=========================================================================*)

FUNCTION bgSSMInitWbr : UDINT (*Init state machine. MUST be called once, before any other bgSSM function call.*)
	VAR_INPUT
		p : bgSSM_typ;
		pfunInitState : UDINT;
		pfunInterrupt : UDINT;
		pfunCyclicCallback : UDINT;
	END_VAR
END_FUNCTION

FUNCTION bgSSMInit : UDINT (*Init state machine. MUST be called once, before any other bgSSM function call.*)
	VAR_INPUT
		p : bgSSM_typ;
		pfunGetStateName : UDINT;
		pfunCyclicCallback : UDINT;
	END_VAR
END_FUNCTION

FUNCTION bgSSMCyclic : UDINT (*State machine cyclic operation.*)
	VAR_INPUT
		p : bgSSM_typ;
	END_VAR
END_FUNCTION

FUNCTION bgSSMStateNextWithWatchdog : UDINT (*Set SM next state w. timer delay*)
	VAR_INPUT
		p : bgSSM_typ;
		stateNext : UDINT;
		wdogTimeX1ms : UDINT;
	END_VAR
END_FUNCTION

FUNCTION bgSSMStateNextTimeDelay : UDINT (*Set SM next state w. timer delay*)
	VAR_INPUT
		p : bgSSM_typ;
		stateNext : UDINT;
		timeDelayX1ms : UDINT;
	END_VAR
END_FUNCTION

FUNCTION bgSSMStateNextCycleDelay : UDINT (*Set SM next state w. cycles delay*)
	VAR_INPUT
		p : bgSSM_typ;
		stateNext : UDINT;
		delayCycles : UDINT;
	END_VAR
END_FUNCTION

FUNCTION bgSSMStateAfterSub : UDINT (*WBR:  Set SM next state after running subroutine states.*)
	VAR_INPUT
		p : bgSSM_typ;
		stateAfterSub : UDINT;
	END_VAR
END_FUNCTION

FUNCTION bgSSMReturnFromSub : UDINT (*WBR:  Set SM to stateAfterSub state.*)
	VAR_INPUT
		p : bgSSM_typ;
	END_VAR
END_FUNCTION

FUNCTION bgSSMStateNext : UDINT (*Set SM next state.*)
	VAR_INPUT
		p : bgSSM_typ;
		stateNext : UDINT;
	END_VAR
END_FUNCTION

FUNCTION bgSSMIsStateInit : BOOL (*Check if first scan within the current state.*)
	VAR_INPUT
		p : bgSSM_typ;
	END_VAR
END_FUNCTION

FUNCTION bgSSMPrintLogMessage : UDINT (*Check if first scan within the current state.*)
	VAR_INPUT
		p : bgSSM_typ;
	END_VAR
END_FUNCTION

FUNCTION bgSSMPrintToTextLogIEC : UDINT (*Check if first scan within the current state.*)
	VAR_INPUT
		p : bgSSM_typ;
		message : STRING[BGSSM_MESSAGE_LENGTH_IEC];
	END_VAR
END_FUNCTION

FUNCTION bgSSMPrintLogMessageToLogbook : DINT (*Check if first scan within the current state.*)
	VAR_INPUT
		p : bgSSM_typ;
		logIdent : UDINT;
	END_VAR
END_FUNCTION

FUNCTION bgSSMPrintToLogbookIEC : DINT (*Check if first scan within the current state.*)
	VAR_INPUT
		p : bgSSM_typ;
		message : STRING[BGSSM_MESSAGE_LENGTH_IEC];
		logIdent : UDINT;
	END_VAR
END_FUNCTION

FUNCTION bgSSMGetState : UDINT (*Get current SM state*)
	VAR_INPUT
		p : bgSSM_typ;
	END_VAR
END_FUNCTION

FUNCTION bgSSMGetStateText : STRING[32] (*Get current SM state name*)
	VAR_INPUT
		p : bgSSM_typ;
	END_VAR
END_FUNCTION
(*=========================================================================*)
(*SUPPORT FOR FIFOs*)
(*=========================================================================*)

FUNCTION bgFIFOInit : UDINT (*Init simple FIFO. Stores upto (entryTotalCount) number of elements. Elements MUST be of the same size.*)
	VAR_INPUT
		p : bgFIFO_typ;
		entrySize : UDINT;
		entryTotalCount : UDINT;
		pFIFOmem : UDINT;
	END_VAR
END_FUNCTION

FUNCTION bgFIFOPush : UDINT (*Push data to FIFO. Content from pSrc is copied into the available FIFO memory. In case of error return value is != 0*)
	VAR_INPUT
		p : bgFIFO_typ;
		pSrc : UDINT;
		srcSize : UDINT;
	END_VAR
END_FUNCTION

FUNCTION bgFIFOPull : UDINT (*Pull (retrive) data from FIFO. Oldest entry from FIFO memory is copied into the provided pDst space. In case of error return value is != 0*)
	VAR_INPUT
		p : bgFIFO_typ;
		pDst : UDINT;
		dstSize : UDINT;
	END_VAR
END_FUNCTION

FUNCTION bgFIFOGetCount : UDINT (*Get number of entries stored in the FIFO*)
	VAR_INPUT
		p : bgFIFO_typ;
	END_VAR
END_FUNCTION

FUNCTION bgFIFOIsFull : UDINT (*Check if FIFO is full*)
	VAR_INPUT
		p : bgFIFO_typ;
	END_VAR
END_FUNCTION
(*=========================================================================*)
(*Support for TIMERs*)
(*=========================================================================*)

FUNCTION bgTimerOffCyclic : UDINT (*Timer cyclic function. Must be called cyclicly for corret timer operation.*)
	VAR_INPUT
		pTOF : TOF;
	END_VAR
END_FUNCTION

FUNCTION bgTimerCyclic : UDINT (*Timer cyclic function. Must be called cyclicly for corret timer operation.*)
	VAR_INPUT
		pTON : TON;
	END_VAR
END_FUNCTION

FUNCTION bgTimerStart : UDINT (*Start timer for a defined amount of time [ms]. IMPORTANT: function uses TON library call. Same restrictions apply!*)
	VAR_INPUT
		pTON : TON;
		timeoutTimeX1ms : UDINT;
	END_VAR
END_FUNCTION

FUNCTION bgTimerStop : UDINT (*Stop the timer.*)
	VAR_INPUT
		pTON : TON;
	END_VAR
END_FUNCTION

FUNCTION bgTimerIsEnabled : BOOL (*Check if timer is enabled.*)
	VAR_INPUT
		pTON : TON;
	END_VAR
END_FUNCTION

FUNCTION bgTimerIsTimeOut : BOOL (*Check if timer has expired.*)
	VAR_INPUT
		pTON : TON;
	END_VAR
END_FUNCTION

FUNCTION bgTimerTimeElapsed : UDINT (*Retrive the elapsed timer time [ms]*)
	VAR_INPUT
		pTON : TON;
	END_VAR
END_FUNCTION

FUNCTION bgTimerTimeRemaining : UDINT (*Retrive the remainig timer time [ms]*)
	VAR_INPUT
		pTON : TON;
	END_VAR
END_FUNCTION
```

#### bgssm.c
```c
/********************************************************************
 * COPYRIGHT -- belgor
 ********************************************************************
 * Library: bglibas
 * File: bglibas.c
 * Author: admin
 * Created: March 07, 2012
 ********************************************************************
 * Implementation of library bglibas
 ********************************************************************/

#ifdef __cplusplus
  extern "C"
  {
#endif

#include <string.h>
#include <stdarg.h>

#include  "bglibasWBR.h"                                                        //  WBR: could also keep the bglibas.h name and change the library's Properties->Library setting away from using the default name
#include  "bglibasWBR_C.h"

/* Init state machine. MUST be called once, before any other bgSSM function call. */
unsigned long bgSSMInit(struct bgSSM_typ* p, unsigned long pFunGetStateName, unsigned long pFunCyclicCallback)
{
  memset(p, 0, sizeof(struct bgSSM_typ));

  p->pfunGetStateName = (UDINT)pFunGetStateName;
  p->pfunCyclicCallback = (UDINT)pFunCyclicCallback;
  p->stateInit = 1;
  return(0);
}

/** Function pointer Init state machine. MUST be called once, before any other bgSSM function call. */
unsigned long bgSSMInitWbr(struct bgSSM_typ* p,                                    //  Pointer to state machine members and methods
                           unsigned long pfunInitState,                            //  Mandatory - initial method must be assigned
                           unsigned long pfunInterrupt,                            //  Optional
                           unsigned long pFunCyclicCallback)                       //  Optional
{
  memset(p, 0, sizeof(struct bgSSM_typ));

  p->pfunInitState=       (UDINT)pfunInitState;
  p->pfunInterrupt=       (UDINT)pfunInterrupt;
  p->pfunCyclicCallback=  (UDINT)pFunCyclicCallback;

  p->log.str.list=  (linkedList_typ *)listSvcRequestList(BGSSM_MESSAGE_LENGTH_C,  lsQUEUE);

  p->stateNext= p->pfunInitState;                                                   //  WBR: assign init state function

  return(0);
}

/** State machine (SM) cyclic operation. */
unsigned long bgSSMCyclic(struct bgSSM_typ* p)
{
  int ii;

  //  TODO: implement interrupt/pause here to pause the delays with the SM

  //operate all timers
  for(ii=0; ii<BGSSM_TIMER_COUNT;ii++){
    bgTimerCyclic(&p->timer_x1ms[ii]);
  }
  bgTimerCyclic(&p->dlytimer_x1ms);
  bgTimerCyclic(&p->wdogTimer_x1ms);

  if(p->dlyCycles){
    p->dlyCycles--;
  }

  //call cyclic callback function if defined
  if(p->pfunCyclicCallback){
    void(*callback)(bgSSM_typ*) = ( void (*) (bgSSM_typ*) ) p->pfunCyclicCallback;
    (*callback)(p);
  }

  //clear single cycle flag every scan
  p->stateInit = 0;

  /// Evaluate breakpoint feature
  if(p->scanLimit.breakpoint && !p->scanLimit.active)   p->scanLimit.active=  1;          //  breakpoint has been found
  if(p->scanLimit.breakpointPrev && !p->scanLimit.breakpoint)   p->scanLimit.active=  0;  //  breakpoint switched off by

  /// Evaluate limit scan feature
  if(p->scanLimit.triggerNextScan)
  {
    p->scanLimit.triggerNextScan= p->scanLimit.count= 0;
  }
  if(!p->scanLimit.active)          memset(&p->scanLimit, 0, sizeof(p->scanLimit));
  else
  {
    if(p->scanLimit.count >= p->scanLimit.limit)   return 1;
    p->scanLimit.count++;
  }

  //check if state change requested
  if(p->state != p->stateNext){

    //if state change w. delay > wait for delay timer to expire or dlyCycles == 0
    if(!bgTimerIsTimeOut(&p->dlytimer_x1ms) || p->dlyCycles){                   //  TODO: add delay until event?
      return 1;
    }

    p->state = p->stateNext;
    //generate stateInit single scan flag
    p->stateInit = 1;

    //define state name if external function for state names is defined
    if( p->pfunGetStateName ){
      char*(*getStateName)(UDINT) = ( char* (*) (UDINT) )p->pfunGetStateName;
      strcpy(p->stateText, (*getStateName)(p->state));
    }else{
      strcpy(p->stateText, "???");
    }
  }

  if(p->pfunInitState)                                                          //  if the init state function pointer is defined...
  {
    void(*callState)(bgSSM_typ*) = ( void (*) (bgSSM_typ*) ) p->state;          //  ... call the function for the current state, i.e. use function pointer SM - WBR:
    (*callState)(p);
  }
  return(0);
}

/** SM state change methods
=============================*/

/** Change to next state. */
unsigned long bgSSMStateNext(struct bgSSM_typ* p, unsigned long stateNext)
{
  p->stateNext = stateNext;
  return(p->stateNext);
}

/** Store state to go to after SM subroutine. */
unsigned long bgSSMStateAfterSub(struct bgSSM_typ* p, unsigned long stateAfterSub)
{
  if(p->stateAfterSubIndex >= BGSSM_SUBROUTINE_COUNT)   return -99;     //  TODO: handle this error

  p->stateAfterSub[p->stateAfterSubIndex] = stateAfterSub;
  return(p->stateAfterSub[p->stateAfterSubIndex++]);
}

/** Activate state to go to after SM subroutine. */
unsigned long bgSSMReturnFromSub(struct bgSSM_typ* p)
{
  if(p->stateAfterSubIndex >= BGSSM_SUBROUTINE_COUNT)   return -99;     //  TODO: handle this error

  p->stateNext=    p->stateAfterSub[p->stateAfterSubIndex--];
  return(p->stateNext);
}

/** Change to next state w. timer delay. */
unsigned long bgSSMStateNextWithWatchdog(struct bgSSM_typ* p, unsigned long stateNext, unsigned long wdogTimeX1ms)
{
  p->stateNext = stateNext;
  bgTimerStart(&p->wdogTimer_x1ms, wdogTimeX1ms);
  return(p->stateNext);
}

/** Change to next state w. timer delay. */
unsigned long bgSSMStateNextTimeDelay(struct bgSSM_typ* p, unsigned long stateNext, unsigned long delayTimeX1ms)
{
  p->stateNext = stateNext;
  bgTimerStart(&p->dlytimer_x1ms, delayTimeX1ms);
  return(p->stateNext);
}

/** Change to next state w. cycles delay. */
unsigned long bgSSMStateNextCycleDelay(struct bgSSM_typ* p, unsigned long stateNext, unsigned long delayCycles)
{
  p->stateNext = stateNext;
  p->dlyCycles = delayCycles;
  return(p->stateNext);
}

/** Check if first scan for the state. */
plcbit bgSSMIsStateInit(struct bgSSM_typ* p)
{
  return(p->stateInit);
}

/** \todo  document */
UDINT  bgSSMPrintToTextLog(struct bgSSM_typ* p, const char* format, ...)
{
 va_list ap;

  va_start(ap, format);
  wbrvsnprintf((char *)listSvcRequestListNode(p->log.str.list), BGSSM_MESSAGE_LENGTH_C, format, ap);
  va_end(ap);

  return  listSvcCharListToStringArray(
                  p->log.str.list
                , &p->log.view[0][0]
                , BGSSM_MESSAGE_LENGTH_C
                , BGSSM_LOG_ENTRIES
                , p->log.str.i.offset
                , p->log.str.i.pageOffset
                , 1
                , ""
               );
}

/** \todo  document */
UDINT  bgSSMPrintLogMessage(struct bgSSM_typ* p)
{
  return  bgSSMPrintToTextLog(p, "%s", p->msg.log);
}

/** \todo  document */
UDINT  bgSSMPrintToTextLogIEC(struct bgSSM_typ* p, char* message)
{
  return  bgSSMPrintToTextLog(p, "%s", message);
}

/** \todo  document */
DINT  bgSSMPrintToLogbook(struct bgSSM_typ* p, const char* text, UDINT logIdent)
{
  return  requestMessageToLog( (UDINT)text, logIdent, 0, 0, 0, 0);              //  logIdent currently not used if logMsgType param is zero
}

/** \todo  document */
DINT  bgSSMPrintLogMessageToLogbook(struct bgSSM_typ* p, UDINT logIdent)    //! \todo   strcpy(loggermsg, requestedmsg) since msg gets destroyed, at least in ARsim
{
  return  requestMessageToLog( (UDINT)p->msg.log, logIdent, 0, 0, 0, 0);           //  logIdent currently not used if logMsgType param is zero
}

/** \todo  document */
DINT  bgSSMPrintToLogbookIEC(struct bgSSM_typ* p, char* message, UDINT logIdent)    //! \todo   strcpy(loggermsg, requestedmsg) since msg gets destroyed, at least in ARsim
{
  return  requestMessageToLog( (UDINT)message, logIdent, 0, 0, 0, 0);           //  logIdent currently not used if logMsgType param is zero
}

/** Check if first scan for the state.  If yes, perform some standard state change functions */
//plcbit bgSSMIsStateInitWBR( struct bgSSM_typ* p
//                          , const char* stateText)           //!<  This can take __FUNCTION__ or "text"
//{
//  if(p->stateInit)
//  {
//    if(stateText)  strcpy(p->stateText, stateText);
//    wbrsnprintf(p->msg.log, sizeof(p->msg.log), "%s(%d)", bgSSMGetStateText(p), bgSSMGetState(p));      //! \todone? reserve p->message for other messages?
//    bgSSMPrintToTextLog(p, "%s", p->msg.log);
//    bgSSMPrintToLogbook(p, p->msg.log, 1);
//  }
//
//  return(p->stateInit);
//}

/** SM data retrieval methods
=============================*/

/** Get current state */
unsigned long bgSSMGetState(struct bgSSM_typ* p)
{
  return(p->state);
}

/** Get current state text*/
plcstring* bgSSMGetStateText(struct bgSSM_typ* p)
{
  return(&p->stateText[0]);
}

#ifdef __cplusplus
  };
#endif
```

### Package Logical/Libraries/wbrServices/wbrSvcUtilities - Utility functions

### Library Logical/Libraries/wbrServices/wbrSvcUtilities/wbrFltUtil

#### wbrFltUtil.fun
```iecst
(********************************************************************
 * COPYRIGHT -- Piedmont Automation
 ********************************************************************
 * Library: wbrFltUtil
 * File: wbrFltUtil.fun
 * Author: Blanton Radford
 * Created: August 18, 2015
 ********************************************************************
 * Functions and function blocks of library wbrFltUtil
 ********************************************************************)

FUNCTION wbrDoubleInRange : BOOL (*Checks that the double v1 is between lo and hi*)
	VAR_INPUT
		lo : LREAL;
		v1 : LREAL;
		hi : LREAL;
	END_VAR
END_FUNCTION

FUNCTION wbrDoubleCompare : BOOL (*Compares two doubles ()v1, v2)  to see if they are within the tolerance value (tol)*)
	VAR_INPUT
		v1 : LREAL;
		v2 : LREAL;
		tol : LREAL;
	END_VAR
END_FUNCTION
```

#### wbrFloatUtilities.c
```c
/********************************************************************
 * \copyright -- Piedmont Automation
 ********************************************************************
 * Program : wbrFltUtil
 * \file :   wbrFloatUtilities.c
 * \author : Blanton Radford
 * \date Created: August 18, 2015
 *******************************************************************/

#include <bur/plctypes.h>

BOOL  wbrDoubleInRange(double lo, double v1, double hi)
{
  return  ((lo < v1) && (v1 < hi));
}

BOOL  wbrDoubleCompare(double v1, double v2, double tol)
{
  return  wbrDoubleInRange(v2-tol,  v1,   v2+tol);
}
```

### Package Logical/Libraries/wbrServices/InitSP - Place this program in TC#1 to initialize wbrServices

### Program Logical/Libraries/wbrServices/InitSP/runFirst

#### svninfo.c
```c
char *Revision      = "748";
char *Modified      = "Modified";
char *Date          = "2017/04/12 15:30:38";
char *TimeNow       = "2017/04/13 11:08:24";
char *RevRange      = "745:748";
char *Mixed         = "Mixed revision WC";
char *IsTagged      = "Not tagged";
char *URL           = "http://99.33.108.51/Internal/MarketingAlliance/trunk/software/AriesV2";
char *isInSVN       = "versioned";
char *lockdate      = "1969/12/31 19:00:00";
```

### Program Logical/Application/Creaser (IEC)

#### Main.st - Init, cyclic, exit code
```iecst
PROGRAM _INIT

	Action_Init_Infeed_Axis; //Set pointer values/initialize servo drive FBK MpAxisBasic instance

	MachineState := MACHINE_STATE_INIT;

	Pulse_Slow.TimeOn := DEFINE_SLOW_PULSE_PERIOD;
	Pulse_Slow.TimeOff := DEFINE_SLOW_PULSE_PERIOD;

	Pulse_Fast.TimeOn := DEFINE_FAST_PULSE_PERIOD;
	Pulse_Fast.TimeOff := DEFINE_FAST_PULSE_PERIOD;

END_PROGRAM

PROGRAM _CYCLIC

	IF gStatistics.Reset THEN //Reset all statistics
		brsmemset(ADR(gStatistics), 0, SIZEOF(Global_Statistics_typ)); //Kind of a weird way to do this- essentially just writes 0's to the entirety of the memory the structure occupies (thus "zeroing-out" the counters)
	END_IF;

	Action_Eval_ErrorState_Statuses; //Evaluate the conditions that put machine into ERR state

	//Eval conditions that would send the machine into ERR state if the machine isn't already in ERR or INIT state->

	IF EDGEPOS(IO.iSafeMachineState) OR iMachineErrorReset THEN
		ProcessState := PRCS_STATE_INIT;
		gAlarmResetRequested := TRUE;
		//		gStatistics.Reset := TRUE;
		MachineState := MACHINE_STATE_INIT;
	END_IF;

	IF EDGEPOS(MachineState = MACHINE_STATE_ERROR) THEN
		AxisControl.MoveVelocity := FALSE;
		AxisControl.MoveAbsolute := FALSE;
		AxisControl.MoveAdditive := FALSE;
		AxisControl.Stop := TRUE;
		AxisControl();
	END_IF;

	BoardEjectUIButton_Hide := BOOL_TO_USINT(NOT ((MachineState = MACHINE_STATE_IDLE OR MachineState = MACHINE_STATE_MANUAL_EJECT) AND IO.iFiberOpticSensor));

	StartUIButton_Hide := NOT (MachineState = MACHINE_STATE_IDLE);
	StopUIButton_Hide := NOT (MachineState = MACHINE_STATE_RUNNING);

	CASE MachineState OF
		MACHINE_STATE_INIT:
			IO.oBoardFeedingLight := FALSE;
			IO.oUIIndicatorLight := FALSE;
			AxisControl.Power := FALSE;

			MachineState := MACHINE_STATE_HARDWARE_INIT;

		MACHINE_STATE_HARDWARE_INIT:
			IO.oBoardFeedingLight := FALSE;
			IO.oUIIndicatorLight := FALSE;

			IF AxisControl.Info.ReadyToPowerOn THEN
				AxisControl.Power := TRUE;
				MachineState := MACHINE_STATE_AXIS_POWER;
			END_IF;

		MACHINE_STATE_AXIS_POWER:
			IO.oBoardFeedingLight := FALSE;
			IO.oUIIndicatorLight := FALSE;

			IF AxisControl.PowerOn THEN
				Action_Stop_Feeder;
				MachineState := MACHINE_STATE_IDLE;
			END_IF;

		MACHINE_STATE_IDLE:
			IO.oBoardFeedingLight := FALSE;
			IO.oUIIndicatorLight := Pulse_Slow.bFlashOut;

			IF EDGEPOS(iManualBoardEject) THEN

				AxisControl.MoveVelocity := FALSE;
				AxisControl.MoveAbsolute := FALSE;
				AxisControl.MoveAdditive := FALSE;
				AxisControl.Stop := FALSE;
				AxisControl();

				AxisPar.Velocity := gRecCfg.active.Rec.FeedVelocity;
				AxisPar.Acceleration := gRecCfg.active.Cfg.Creaser.FeedAxisAccel;
				AxisPar.Deceleration := gRecCfg.active.Cfg.Creaser.FeedAxisDecel;

				AxisControl.MoveVelocity := TRUE;
				AxisControl();

				MachineState := MACHINE_STATE_MANUAL_EJECT;
			END_IF;

			IF EDGEPOS(iStartCommand) THEN
				IF IO.iFiberOpticSensor THEN
					gAlarms.Fiber_Optic_Blocked_RunCmd := TRUE;
					MachineState := MACHINE_STATE_ERROR;
				ELSIF NOT IO.iCreaserShaftSensor THEN
					gAlarms.Manual_Home_Creaser_Blade := TRUE;
					MachineState := MACHINE_STATE_ERROR;
				ELSE
					//					setflagCreaserIndexCommand := TRUE;
					iSoftStopCommand := FALSE;
					Action_Start_Feeder;
					ProcessState := PRCS_STATE_INIT;
					MachineState := MACHINE_STATE_RUNNING;
				END_IF;
			END_IF;

		MACHINE_STATE_MANUAL_EJECT:
			IO.oBoardFeedingLight := TRUE;
			IO.oUIIndicatorLight := Pulse_Slow.bFlashOut;

			IF (NOT IO.iFiberOpticSensor AND IO_LastCycle.iFiberOpticSensor) OR NOT iManualBoardEject THEN
				Action_Stop_Feeder;
				MachineState := MACHINE_STATE_IDLE;
			END_IF;

		MACHINE_STATE_RUNNING:
			IO.oUIIndicatorLight := TRUE;

			Action_Manage_Update_Total_Runtime;

			Action_Tally_Board_L;

			IF iSoftStopCommand THEN

				IF NOT (ProcessState = PRCS_STATE_SOFT_STOP) THEN
					Action_Stop_Feeder;
				END_IF;

				ProcessState := PRCS_STATE_SOFT_STOP;
			END_IF;

			Action_CreaserProcess_SM; //Crease motor <-> movement cycle <-> FiOS state machine

		MACHINE_STATE_ERROR: //ERROR state.  Note that this state is exited via the logic ABOVE the state machine.
			IO.oBoardFeedingLight := FALSE;
			IO.oUIIndicatorLight := Pulse_Fast.bFlashOut AND Pulse_Slow.bFlashOut;

			Current_Crease_Section_Length := 0;

			ProcessState := PRCS_STATE_INIT;

	END_CASE;

	Pulse_Slow;
	Pulse_Fast;

	Action_Creaser_Idx; //Reads/sets flag variables indicating current state of the creasing motor
	Action_AxisControl_Mgmt; //Calls Infeed Axis Control FBK, sets/resets drive errors

	IO_LastCycle := IO; //Latch previous cycle IO values (since EDGEPOS() has some weird caveats)
END_PROGRAM

PROGRAM _EXIT
	(* Insert code here *)

END_PROGRAM
```

#### Variables.var - Local variables
```iecst
VAR
	Timer_Creaser_Idx_Edge : TON;
	Timer_Total_Runtime : TON;
	tmp_bool : BOOL;
	setFlagTravelEdgeOffset : BOOL;
	setFlagCreaserIdxFinished : BOOL;
	setflagCreaserIndexCommand : BOOL;
	setStartCommandFlag : BOOL;
	setFlagCreaserIndexed : BOOL;
	setFlagCreaserWaitEdge : BOOL;
END_VAR
```

#### Action_Start_Feeder.st
```iecst
ACTION Action_Start_Feeder:
	AxisControl.MoveVelocity := FALSE;
	AxisControl.MoveAbsolute := FALSE;
	AxisControl.MoveAdditive := FALSE;
	AxisControl.Stop := FALSE;
	AxisControl();

	AxisPar.Velocity := gRecCfg.active.Cfg.Creaser.PreInsertSpeed;
	AxisPar.Acceleration := gRecCfg.active.Cfg.Creaser.FeedAxisAccel;
	AxisPar.Deceleration := gRecCfg.active.Cfg.Creaser.FeedAxisDecel;

	AxisControl.MoveVelocity := TRUE;
	AxisControl();
END_ACTION
```

#### Action_Move_Section_Distance.st
```iecst
ACTION Action_Move_Section_Distance:

	AxisControl.MoveAbsolute := FALSE;
	AxisControl.MoveAdditive := FALSE;
	AxisControl.MoveVelocity := FALSE;
	AxisControl.Stop := FALSE;
	AxisControl();

	Current_Crease_Section_Length := gRecCfg.active.Rec.Crease.CreaseDistance_mm[ii_crease_count];

	AxisPar.Acceleration := gRecCfg.active.Cfg.Creaser.FeedAxisAccel;
	AxisPar.Deceleration := gRecCfg.active.Cfg.Creaser.FeedAxisDecel;
	AxisPar.Distance := gRecCfg.active.Rec.Crease.CreaseDistance_mm[ii_crease_count];
	AxisPar.Velocity := gRecCfg.active.Rec.FeedVelocity;

	AxisControl.MoveAdditive := TRUE;
	AxisControl();

END_ACTION
```

#### Action_Creaser_Idx.st
```iecst
ACTION Action_Creaser_Idx:

		//Temp. Sim. code->

	IF gSimulateMachine THEN
		Timer_Sim_CreaserIdx.PT := T#500ms;
		Timer_Sim_CreaserIdx.IN := setFlagCreaserWaitEdge;
		Timer_Sim_CreaserIdx();
		IO.iCreaserShaftSensor := Timer_Sim_CreaserIdx.Q;
	END_IF;

	setFlagCreaserIdxFinished := FALSE;

	IF setflagCreaserIndexCommand THEN
		setFlagTravelEdgeOffset := FALSE;
		setFlagCreaserWaitEdge := TRUE;
	END_IF;

	IF setFlagCreaserWaitEdge THEN
		IO.oCreaserCCWRotation := (gRecCfg.active.Rec.Crease.CreaserDirection = 0);
		IO.oCreaserCWRotation  := (gRecCfg.active.Rec.Crease.CreaserDirection = 1);

		IF setFlagTravelEdgeOffset AND bgTimerIsTimeOut(Timer_Creaser_Idx_Edge) THEN
			setFlagTravelEdgeOffset := FALSE;
			setFlagCreaserWaitEdge := FALSE;
			setFlagCreaserIdxFinished := TRUE;

			gStatistics.total_creases := gStatistics.total_creases + 1;
		END_IF;

		CASE gRecCfg.active.Rec.Crease.ShaftSensorEdge OF
			0:
				IF IO.iCreaserShaftSensor AND NOT IO_LastCycle.iCreaserShaftSensor AND NOT setFlagTravelEdgeOffset THEN
					setFlagTravelEdgeOffset := TRUE;
					bgTimerStart(Timer_Creaser_Idx_Edge, Tms(gRecCfg.active.Rec.Crease.CreaserMotorIdxLag_S));
				END_IF;
			1:
				IF NOT IO.iCreaserShaftSensor AND IO_LastCycle.iCreaserShaftSensor AND NOT setFlagTravelEdgeOffset THEN
					setFlagTravelEdgeOffset := TRUE;
					bgTimerStart(Timer_Creaser_Idx_Edge, Tms(gRecCfg.active.Rec.Crease.CreaserMotorIdxLag_S));
				END_IF;
		END_CASE;
	ELSE
		IO.oCreaserCCWRotation := FALSE;
		IO.oCreaserCWRotation  := FALSE;
	END_IF;

	bgTimerCyclic(Timer_Creaser_Idx_Edge);

	setflagCreaserIndexCommand := FALSE;
END_ACTION
```

#### Action_AxisControl_Mgmt.st
```iecst
ACTION Action_AxisControl_Mgmt:

	IF EDGEPOS(iMachineErrorReset) THEN
		AxisControl.ErrorReset := TRUE;
	ELSIF EDGENEG(iMachineErrorReset)  THEN
		AxisControl.ErrorReset := FALSE;
	END_IF;

	IF AxisControl.ErrorReset AND NOT AxisControl.Error THEN //FBK errors only reset on + edge of error reset signal -> Clear reset signal when there are no errors!
		AxisControl.ErrorReset := FALSE;
	END_IF;

	Axis1; //Reference the PV cyclically to ensure it registers as being included in the program!
	AxisControl();//Call the function block responsible for executing the axis commands

END_ACTION
```

#### Action_Move_Crease_Width.st
```iecst
ACTION Action_Move_Crease_Width:
	AxisControl.MoveVelocity := FALSE;
	AxisControl.MoveAbsolute := FALSE;
	AxisControl.MoveAdditive := FALSE;
	AxisControl.Stop := FALSE;
	AxisControl();

	AxisPar.Acceleration := gRecCfg.active.Cfg.Creaser.FeedAxisAccel;
	AxisPar.Deceleration := gRecCfg.active.Cfg.Creaser.FeedAxisDecel;
	AxisPar.Distance := 	gRecCfg.active.Rec.Crease.CreaseWidth_mm;
	AxisPar.Velocity := gRecCfg.active.Rec.FeedVelocity;

	AxisControl.MoveAdditive := TRUE;
	AxisControl();
END_ACTION
```

#### Action_CreaserProcess_SM.st - not listed in the package file held
```iecst
ACTION Action_CreaserProcess_SM:

	CASE ProcessState OF
		PRCS_STATE_INIT:
			IO.oBoardFeedingLight := FALSE;
			Current_Board_Position := 0;
			iSoftStopCommand := FALSE;

			Action_Validate_Board_Length;

			IF flagBoardLengthCfgErr AND (gRecCfg.active.Cfg.Creaser.BypassBoardLengthError = 0) THEN
				flagBoardLengthCfgErr := FALSE;
				ProcessState := PRCS_STATE_ERROR;
			ELSIF IO.iCreaserShaftSensor THEN
				ii_crease_count := 0;
				ProcessState := PRCS_STATE_READY;
			END_IF;

		PRCS_STATE_READY:
			IO.oBoardFeedingLight := FALSE;
			Current_Board_Position := 0;

			IF AxisControl.InVelocity THEN
				ii_crease_count := 0;
				ProcessState := PRCS_STATE_FEED_BOARD;
			END_IF;

		//				PRCS_STATE_FEED_BOARD:
		//					IO.oBoardFeedingLight := TRUE;
		//					IF IO.iFiberOpticSensor AND NOT IO_LastCycle.iFiberOpticSensor THEN
		//						Action_Move_Section_Distance;
		//
		//						Current_Board_Position := 0;
		//
		//						ProcessState := PRCS_STATE_MOVE_CREASE;
		//					END_IF;

		PRCS_STATE_FEED_BOARD:
			IO.oBoardFeedingLight := TRUE;

			Current_Board_Position := 0;

			IF IO.iFiberOpticSensor AND NOT IO_LastCycle.iFiberOpticSensor THEN
				Action_Move_Photoeye_Offset;

				ProcessState := PRCS_STATE_MOVE_PHOTOEYE_OFFSET;
			END_IF;

		PRCS_STATE_MOVE_PHOTOEYE_OFFSET:
			IO.oBoardFeedingLight := Pulse_Slow.bFlashOut;

			IF AxisControl.InPosition THEN
				Action_Move_Section_Distance;
				Current_Board_Position := 0;
				ProcessState := PRCS_STATE_MOVE_CREASE;
			END_IF;

		PRCS_STATE_MOVE_CREASE:
			IO.oBoardFeedingLight := Pulse_Slow.bFlashOut;
			IF AxisControl.InPosition THEN
				setflagCreaserIndexCommand := TRUE;
				ProcessState := PRCS_STATE_CREASE;
			END_IF;

		PRCS_STATE_CREASE:
			IO.oBoardFeedingLight := Pulse_Fast.bFlashOut;

			IF setFlagCreaserIdxFinished THEN //Wait for flag set by creaser that it has indexed and is at the "ready" position to move board
				ii_crease_count := ii_crease_count + 1; //Increment crease counter

				IF ii_crease_count = (gRecCfg.active.Rec.Crease.CreaseCount) THEN
					//							Action_Start_Feeder;

					AxisControl.MoveVelocity := FALSE;
					AxisControl.MoveAbsolute := FALSE;
					AxisControl.MoveAdditive := FALSE;
					AxisControl.Stop := FALSE;
					AxisControl();

					AxisPar.Velocity := gRecCfg.active.Rec.FeedVelocity;
					AxisPar.Acceleration := gRecCfg.active.Cfg.Creaser.FeedAxisAccel;
					AxisPar.Deceleration := gRecCfg.active.Cfg.Creaser.FeedAxisDecel;

					AxisControl.MoveVelocity := TRUE;
					AxisControl();

					ProcessState := PRCS_STATE_EJECT_FINISHED_BOARD;
				ELSE
					Action_Move_Crease_Width;
					ProcessState := PRCS_STATE_MOVE_CREASE_WIDTH;
				END_IF;
			END_IF;

		PRCS_STATE_MOVE_CREASE_WIDTH:
			IO.oBoardFeedingLight := Pulse_Slow.bFlashOut;

			IF AxisControl.InPosition THEN
				Action_Move_Section_Distance;
				ProcessState := PRCS_STATE_MOVE_CREASE;
			END_IF;

		PRCS_STATE_EJECT_FINISHED_BOARD:
			IO.oBoardFeedingLight := Pulse_Slow.bFlashOut AND Pulse_Fast.bFlashOut;

			IF NOT IO.iFiberOpticSensor AND IO_LastCycle.iFiberOpticSensor THEN

				Latch_Board_Length := Current_Board_Position + gRecCfg.active.Cfg.Creaser.PhotoEyeOffset;

				IF (Latch_Board_Length > (gRecCfg.active.Rec.Crease.TotalBoardLength + gRecCfg.active.Cfg.Creaser.BoardLengthTolerance)) AND (gRecCfg.active.Cfg.Creaser.BypassBoardLengthError = 0) THEN
					gAlarms.Measured_Length_GT_Configured := TRUE;
					ProcessState := PRCS_STATE_ERROR;
				ELSIF (Latch_Board_Length < (gRecCfg.active.Rec.Crease.TotalBoardLength - gRecCfg.active.Cfg.Creaser.BoardLengthTolerance)) AND (gRecCfg.active.Cfg.Creaser.BypassBoardLengthError = 0) THEN
					gAlarms.Measured_Length_LT_Configured := TRUE;
					ProcessState := PRCS_STATE_ERROR;
				ELSE
					gStatistics.total_processed := gStatistics.total_processed + 1;
					gStatistics.Sum_Board_Travel_Lengths := gStatistics.Sum_Board_Travel_Lengths + Latch_Board_Length;
					gStatistics.Avg_Board_Length := gStatistics.Sum_Board_Travel_Lengths / UDINT_TO_REAL(gStatistics.total_processed);

					Action_Start_Feeder;

					ProcessState := PRCS_STATE_READY;
				END_IF;

			END_IF;

		PRCS_STATE_ERROR:
			IO.oBoardFeedingLight := FALSE;

		PRCS_STATE_SOFT_STOP:
			IO.oBoardFeedingLight := FALSE;

			IF NOT iSoftStopCommand THEN
				Action_Start_Feeder;

				IF IO.iFiberOpticSensor THEN  //Eject this part, maybe in the future resume from last state but for now just consider the current part a wash
					ProcessState := PRCS_STATE_INIT;
				ELSE //Re-cycle back to process SM jump-off point
//					setflagCreaserIndexCommand := TRUE;
					ii_crease_count := 0;
					ProcessState := PRCS_STATE_INIT;
				END_IF;
			END_IF;
	END_CASE;

END_ACTION
```

#### Action_Transition_Feed_Vel_Additive.st - not listed in the package file held
```iecst
ACTION Action_Transition_Feed_Vel_Additive:

END_ACTION
```

### Library Logical/Application/Dispense/libValve (IEC)
Depends on: libAS52XX

#### FBK_Hernon_SureShot.st
```iecst
(* TODO: Add your comment here *)
FUNCTION_BLOCK FBK_Hernon_SureShot

	IF iReset THEN
		iReset := FALSE;
		brsmemset(ADR(Alarms), 0, SIZEOF(HERNON_Alarm_Dispense_typ));
		oState := DISPENSE_STATE_INIT;
	END_IF;

//The following shows the archetypal logic for what happens when the valve BECOMES disabled/deactivated-
//	IF (Config.Disable = 1) AND NOT (oState = DISPENSE_STATE DISABLED OR oState = DISPENSE_STATE_INIT) THEN
//		//Valve was disabled
//	ELSIF (Config.Disable = 0 AND Recipe.Enable = 0) AND NOT (oState = DISPENSE_STATE INACTIVE OR oState = DISPENSE_STATE_INIT) THEN
//		//Valve was deactivated
//	END_IF;

	IF NOT IO.EdgeGen.iEdgeGenError THEN
		IO.EdgeGen.oQuitEdgeGenError := FALSE;
	END_IF;

	IF NOT IO.EdgeGen.iEdgeGenWarning THEN
		IO.EdgeGen.oQuitEdgeGenWarning := FALSE;
	END_IF;

	Alarms.EdgeGenError := IO.EdgeGen.iEdgeGenError;

	IO.EdgeGen.oEdgeGenOffset := Tms(Recipe.Disp_Valve_Edgemode_Pulse_TO_ms);

	CASE oState OF
		DISPENSE_STATE_INIT:
			oHMIColorDP := HMI_PRCS_COLOR_DISABLED;

			IO.oDispTrigger := FALSE;
			iFlagDispenseNow := FALSE;
			ii_shot_counter := 0;
			IO.EdgeGen.oEnableEdgeGen := TRUE;

			//Following conditionals are for the X20DS4389 unit to ACK the error bit on the IO modules if it is set (only in INIT state of the valve)
			IF IO.EdgeGen.iEdgeGenError AND IO.EdgeGen.oQuitEdgeGenError THEN
				IO.EdgeGen.oQuitEdgeGenError := TRUE;
			ELSE
				IO.EdgeGen.oQuitEdgeGenError := FALSE;
			END_IF;

			IF IO.EdgeGen.iEdgeGenWarning AND IO.EdgeGen.oQuitEdgeGenWarning THEN
				IO.EdgeGen.oQuitEdgeGenWarning := TRUE;
			ELSE
				IO.EdgeGen.oQuitEdgeGenWarning := FALSE;
			END_IF;

			(*IF Config.Disable = 1 THEN*)
				IF Recipe.Enable = 0 THEN
					oState := DISPENSE_STATE_INACTIVE;
				ELSIF (IO.iValveReady AND NOT IO.EdgeGen.iEdgeGenError) THEN
					oState := DISPENSE_STATE_READY;
				END_IF;
//			ELSIF (IO.iValveReady AND NOT IO.EdgeGen.iEdgeGenError) THEN
//				oState := DISPENSE_STATE_READY;
//			END_IF;

		DISPENSE_STATE_READY:
			oHMIColorDP := HMI_PRCS_COLOR_IDLE;

			IF Recipe.Enable = 0 THEN
				oState := DISPENSE_STATE_INACTIVE;
			ELSIF (NOT IO.iValveReady OR IO.EdgeGen.iEdgeGenError) THEN
				//				pDispVBlock.Error.DispenseValveError := TRUE;
				//				gAlarms.Dispense.Valve_Error_1[ii_dispense_units] := TRUE;

				Alarms.Valve_Not_Ready := TRUE;

				oState := DISPENSE_STATE_ERROR;
			ELSIF iFlagDispenseNow THEN
				ii_shot_counter := 0;
				IO.oDispTrigger := TRUE;

				IO.EdgeGen.oEdgeGenTimestamp := iX2XNettime + DEFINE_TK_CYCLE_OFFSET;//Immediately give the DS card the timestamp to turn the valve off
				IO.EdgeGen.oEdgeGenSequence := IO.EdgeGen.oEdgeGenSequence + 1;//Incrementing the edge gen sequence number is what causes the new timestamp to take hold (otherwise, it would trigger every time the clock rolls over)

				iFlagDispenseNow := FALSE;
				iFlagDispenseOnFractionOffset := FALSE;
				oDispenseMode := DISPENSE_SINGLE_SHOT;
				oState := DISPENSE_STATE_DISPENSING;
			ELSIF iFlagPurgeNow THEN
				IO.oDispTrigger := TRUE;

				bgTimerStart(Timers.Max_Dispense_Output_High, PURGE_SOFTWARE_TIME_LIMIT);
//				oEdge_Reading_At_Disp_Trigger := IO.EdgeGen.iEdgeMasterTime;

				oDispenseMode := DISPENSE_PURGE;
				oState := DISPENSE_STATE_DISPENSING;
			ELSIF iFlagDispenseOnFractionOffset THEN
				iFlagDispenseNow := FALSE;
				iFlagDispenseOnFractionOffset := FALSE;
				bgTimerStart(Timers.Max_Fractional_Offset_Wait, MAX_TIME_WAIT_FRACTION_OFFSET);
				oState := STATE_WAIT_FRACTION_OFFSET;
			END_IF;

		STATE_WAIT_FRACTION_OFFSET:
			oHMIColorDP := HMI_PRCS_COLOR_ACTIVE;

			IF (iVBlockFractionalPosition > Recipe.Fractional_Position_Offset AND iVBlockFractionalPosition_old < Recipe.Fractional_Position_Offset) OR Recipe.Fractional_Position_Offset < 0.01 THEN
				ii_shot_counter := 0;
				IO.oDispTrigger := TRUE;

				IO.EdgeGen.oEdgeGenTimestamp := iX2XNettime + DEFINE_TK_CYCLE_OFFSET;//Immediately give the DS card the timestamp to turn the valve off
				IO.EdgeGen.oEdgeGenSequence := IO.EdgeGen.oEdgeGenSequence + 1;//Incrementing the edge gen sequence number is what causes the new timestamp to take hold (otherwise, it would trigger every time the clock rolls over)

				oDispenseMode := DISPENSE_SINGLE_SHOT;
				oState := DISPENSE_STATE_DISPENSING;
			ELSIF bgTimerIsTimeOut(Timers.Max_Fractional_Offset_Wait) THEN
				Alarms.Max_Time_Fractional_Offset := TRUE;
				oState := DISPENSE_STATE_ERROR;
			END_IF;

//		DISPENSE_STATE_WAIT_VALVE:
//			oHMIColorDP := HMI_PRCS_COLOR_ACTIVE;
//
//			IF IO.EdgeGen.iEdgeMasterTime <> oEdge_Reading_At_Disp_Trigger THEN
//				IO.oDispTrigger := FALSE;
//
//				IO.EdgeGen.oEdgeGenTimestamp := IO.EdgeGen.iEdgeMasterTime + Tms(Recipe.Disp_Valve_Edgemode_Pulse_TO_ms);//Tms normally converts S->mS, but here it does ms->us
//				IO.EdgeGen.oEdgeGenSequence := IO.EdgeGen.oEdgeGenSequence + 1;//Incrementing the edge gen sequence number is what causes the new timestamp to take hold (otherwise, it would trigger every time the clock rolls over)
//
////				bgTimerStart(Timers.Max_Time_Disp_Output_NegEdge, REAL_TO_UDINT(Recipe.Disp_Valve_Edgemode_Pulse_TO_ms) + NEG_EDGE_MARGIN);//Timer for maximum amount of time to wait before throwing an error, since the DO is reset via the edge generator and not the IO BOOL datapoint itself
//
//				oState := DISPENSE_STATE_DISPENSING;
//			ELSIF (bgTimerIsTimeOut(Timers.Max_Valve_NotRdy_NegEdge)) AND IO.iValveReady THEN
//				IO.oDispTrigger := FALSE;
//
//
//				IO.EdgeGen.oEdgeGenTimestamp := iX2XNettime + 10000;//
//				IO.EdgeGen.oEdgeGenSequence := IO.EdgeGen.oEdgeGenSequence + 1;//Incrementing the edge gen sequence number is what causes the new timestamp to take hold (otherwise, it would trigger every time the clock rolls over)
//
//				//					gAlarms.Dispense.Dispense_ValveRdy_NegEdge_Err[ii_dispense_units] := TRUE;
//				Alarms.Valve_Ready_Neg_Edge_Error := TRUE;
//				oState := DISPENSE_STATE_ERROR;
//			END_IF;

		DISPENSE_STATE_DISPENSING:

			oHMIColorDP := HMI_PRCS_COLOR_ACTIVE;

			CASE oDispenseMode OF
				DISPENSE_SINGLE_SHOT:
				IF NOT IO.EdgeGen.iReadOutputStatus THEN
					IF ii_shot_counter < Recipe.Extra_Shots_Per_VBlock THEN
						bgTimerStart(Timers.Pause_Additional_Shots, Tms(Recipe.Time_Offset_Additional_Shots));
					END_IF;
					bgTimerStart(Timers.Min_Valve_Rdy_Reset, MIN_SIGNAL_RESET_TO);
					bgTimerStart(Timers.Max_Valve_Rdy_Reset, MAX_SIGNAL_RESET_TO);
					oState := DISPENSE_STATE_WAIT_RESET;
				END_IF;
			DISPENSE_PURGE:
				IO.oDispTrigger := FALSE;
				IF (NOT iFlagPurgeNow) OR bgTimerIsTimeOut(Timers.Max_Dispense_Output_High) THEN
					IO.EdgeGen.oEdgeGenTimestamp := iX2XNettime + 10000;
						IO.EdgeGen.oEdgeGenSequence := IO.EdgeGen.oEdgeGenSequence + 1;

					bgTimerStart(Timers.Min_Valve_Rdy_Reset, MIN_SIGNAL_RESET_TO);
					bgTimerStart(Timers.Max_Valve_Rdy_Reset, MAX_SIGNAL_RESET_TO);
					oState := DISPENSE_STATE_WAIT_RESET;
				END_IF;
			END_CASE;
//
		DISPENSE_STATE_WAIT_RESET://Wait for dispense valve ready to read back TRUE before the SM can go back into ready state, otherwise the rest of the code could trigger it too soon.

			oHMIColorDP := HMI_PRCS_COLOR_ACTIVE;

			IF bgTimerIsTimeOut(Timers.Min_Valve_Rdy_Reset) AND IO.iValveReady AND NOT iFlagPurgeNow THEN
				ii_shot_counter := ii_shot_counter + 1;

				IF ii_shot_counter > Recipe.Extra_Shots_Per_VBlock THEN
					pCyclesCounter := pCyclesCounter + 1;
					oState := DISPENSE_STATE_READY;
				ELSE
					oState := DISPENSE_STATE_WAIT_ADDITIONAL;
				END_IF;

			ELSIF bgTimerIsTimeOut(Timers.Max_Valve_Rdy_Reset) THEN
				Alarms.Valve_Not_Ready := TRUE;
				pCounterValveNotRdy := pCounterValveNotRdy + 1;
				oState := DISPENSE_STATE_READY;
			END_IF;

		DISPENSE_STATE_WAIT_ADDITIONAL:
			oHMIColorDP := HMI_PRCS_COLOR_ACTIVE;

			IF bgTimerIsTimeOut(Timers.Pause_Additional_Shots) THEN
				IO.oDispTrigger := TRUE;

//				oEdge_Reading_At_Disp_Trigger := IO.EdgeGen.iEdgeMasterTime;//Nearly lost my mind to this one, need to document edge reading immediately before triggering output, as the high-speed edge detector has no debounce and it can possibly be a "dirty switch"
				iFlagDispenseNow := FALSE;
				oDispenseMode := DISPENSE_SINGLE_SHOT;

				IO.EdgeGen.oEdgeGenTimestamp := iX2XNettime + DEFINE_TK_CYCLE_OFFSET;//Immediately give the DS card the timestamp to turn the valve off
				IO.EdgeGen.oEdgeGenSequence := IO.EdgeGen.oEdgeGenSequence + 1;//Incrementing the edge gen sequence number is what causes the new timestamp to take hold (otherwise, it would trigger every time the clock rolls over)

				oState := DISPENSE_STATE_DISPENSING;
			END_IF;

		DISPENSE_STATE_INACTIVE:
			oHMIColorDP := HMI_PRCS_COLOR_DISABLED;

			IF Recipe.Enable = 1 THEN
				oState := DISPENSE_STATE_INIT;
			END_IF;

		DISPENSE_STATE_DISABLED:
			oHMIColorDP := HMI_PRCS_COLOR_DISABLED;

			IF Config.Disable = 0 THEN
				oState := DISPENSE_STATE_INIT;
			END_IF;

		DISPENSE_STATE_ERROR://State is exited via the event handler directly above state machine!
			oHMIColorDP := HMI_PRCS_COLOR_FAULT;
	END_CASE;

	iVBlockFractionalPosition_old := iVBlockFractionalPosition;

	//Timer cyclic calls
	bgTimerCyclic(Timers.Max_Valve_Rdy_Reset);
	bgTimerCyclic(Timers.Min_Valve_Rdy_Reset);
	bgTimerCyclic(Timers.Max_Dispense_Output_High);
	bgTimerCyclic(Timers.Pause_Additional_Shots);
	bgTimerCyclic(Timers.Max_Fractional_Offset_Wait);

END_FUNCTION_BLOCK
```

#### ApplicationVariables.typ
```iecst
(*Insert your comment here.*)

TYPE
	HERNON_Disp_AppTimers_typ : 	STRUCT
		Max_Valve_Rdy_Reset : TON;
		Max_Dispense_Output_High : TON;
		Pause_Additional_Shots : TON;
		Max_Fractional_Offset_Wait : TON;
		Min_Valve_Rdy_Reset : TON;
	END_STRUCT;
END_TYPE

(*Insert your comment here.*)
```

#### IO.typ
```iecst
TYPE
	X20DS4389_Edgegen_typ : 	STRUCT
		iEdgeMasterTime : DINT;
		iReadOutputStatus : BOOL;
		oEnableEdgeGen : BOOL;
		iEdgeGenReadbackEnabled : BOOL;
		oEdgeGenSequence : SINT;
		iEdgegenSequenceReadback : SINT;
		oEdgeGenTimestamp : DINT;
		iEdgeGenError : BOOL;
		oQuitEdgeGenError : BOOL;
		iEdgeGenWarning : BOOL;
		oQuitEdgeGenWarning : BOOL;
		iDiffTime : ARRAY[0..1]OF DINT;
		oEdgeGenOffset : UDINT;
	END_STRUCT;
	HERNON_Valve_IOPoint_typ : 	STRUCT
		iValveReady : BOOL;
		oDispTrigger : BOOL;
		EdgeGen : X20DS4389_Edgegen_typ;
	END_STRUCT;
END_TYPE
```

### Auxiliary.var
```iecst
(*Insert your comment here.*)
(*Insert your comment here.*)
VAR CONSTANT
	MAX_IDX_USB_PORTS : USINT := 1;
END_VAR
VAR
	gUSB_Step : USB_Global_SM_Enum := (0);
	USB_Object : ARRAY[0..MAX_IDX_USB_PORTS] OF USB_Object_typ := [(0),2((0))];
END_VAR
VAR CONSTANT
	DEFINE_CONSTANT_MAGIC_PREFIX : UDINT := 16#12345678;
	DEFINE_CONSTANT_MAGIC_SUFFIX : UDINT := 16#87654321;
END_VAR
(*Insert your comment here.*)
VAR RETAIN
	gConfigName : STRING[255];
	gRecipeName : STRING[255];
END_VAR
(*Insert your comment here.*)
(*Insert your comment here.*)
VAR
	Recipe_CSV_Control : MpRecipeCsv := (0);
	Recipe_CSV_Header : MpRecipeCsvHeaderType := (0);
	Recipe_CSV_RegPar : MpRecipeRegPar := (0);
	Recipe_CSV_UI : MpRecipeUI := (0);
	gRecipe_CSV_UIConnect : MpRecipeUIConnectType := (0);
	Alarm_Recipe : MpAlarmBasicUIConnect20Type;
	Alarm_Recipe_UI : MpAlarmBasicUI := (0);
END_VAR
(*Insert your comment here.*)
(*Insert your comment here.*)
VAR
	Config_CSV_Control : MpRecipeCsv := (0);
	Config_CSV_Header : MpRecipeCsvHeaderType := (0);
	Config_CSV_RegPar : MpRecipeRegPar := (0);
	Config_CSV_UI : MpRecipeUI := (0);
	gConfig_CSV_UIConnect : MpRecipeUIConnectType := (0);
	Alarm_Config : MpAlarmBasicUIConnect20Type;
	Alarm_Config_UI : MpAlarmBasicUI := (0);
END_VAR
(*Insert your comment here.*)
(*Insert your comment here.*)
VAR
	File_Manager_Control : MpFileManagerUI := (0);
	File_Manager_UIConnect : MpFileManagerUIConnectType := (0);
	Alarm_File : MpAlarmBasicUIConnect20Type := (0);
	Alarm_File_UI : MpAlarmBasicUI := (0);
END_VAR
(*Insert your comment here.*)
VAR
	Com_Logger_UI : MpComLoggerUI := (0);
	Com_Logger_UIConnect : MpComLoggerUIConnectType := (0);
END_VAR
(*Insert your comment here.*)
(*VAR
	Data_Table_Control : MpDataTableUI;
	Data_Table_UIConnect : MpDataTableUIConnectType;
END_VAR*)
(*Insert your comment here.*)
(*VAR
	Data_Log_Control : MpDataRecorder := (0);
	Data_Log_Header : MpDataRecorderHeaderType := (0);
	Data_Log_Config : MpDataRecorderConfig := (0);
	Data_Log_Config_Struct : MpDataRecorderConfigType := (0);
	Data_Log_RegPar : ARRAY[0..99] OF MpDataRegPar := [100((0))];
END_VAR*)
(*Insert your comment here.*)
VAR
	Alarm_Data : MpAlarmBasicUIConnect20Type := (0);
	Alarm_Data_UI : MpAlarmBasicUI := (0);
END_VAR
```

### Program Logical/Auxiliary_Services_Control/Recipe_Handling

#### Cyclic.st
```iecst
PROGRAM _CYCLIC

	gRecCfg;

	CASE gHmi.prv.currentPage OF
		HMI_RECIPE_20_SELECT:
			pRecCfgUIConnect ACCESS ADR(gRecipe_CSV_UIConnect);
			pCmd ACCESS ADR(loc.Rec.HMI);
		HMI_RECIPE_21_PVLIST:
			pRecCfgUIConnect ACCESS ADR(gRecipe_CSV_UIConnect);
			pCmd ACCESS ADR(loc.Rec.HMI);
		HMI_CONFIG_30_SELECT:
			pRecCfgUIConnect ACCESS ADR(gConfig_CSV_UIConnect);
			pCmd ACCESS ADR(loc.Cfg.HMI);
		HMI_CONFIG_31_PVLIST:
			pRecCfgUIConnect ACCESS ADR(gConfig_CSV_UIConnect);
			pCmd ACCESS ADR(loc.Cfg.HMI);
	END_CASE;

	IF EDGENEG(gHmi.prv.currentPage = HMI_RECIPE_20_SELECT) THEN
		locFindActiveRecipe := 1;
	END_IF;

	IF EDGENEG(gHmi.prv.currentPage = HMI_CONFIG_30_SELECT) THEN
		locFindActiveRecipe := 1;
	END_IF;

	IF loc.Rec.cmd.Copy_default_to_save = 1 THEN
		gRecCfg.save.Rec := gRecCfg.defaultvals.Rec;
	END_IF;

	IF loc.Rec.cmd.Copy_default_to_active = 1 THEN
		gRecCfg.active.Rec := gRecCfg.defaultvals.Rec;
	END_IF;

	IF loc.Rec.cmd.Copy_save_to_active = 1 THEN
		gRecCfg.active.Rec := gRecCfg.save.Rec;
	END_IF;

	IF loc.Rec.cmd.Copy_save_to_default = 1 THEN
		gRecCfg.defaultvals.Rec := gRecCfg.save.Rec;
	END_IF;

	IF loc.Rec.cmd.Copy_active_to_save = 1 THEN
		gRecCfg.save.Rec := gRecCfg.active.Rec;
	END_IF;

	IF loc.Rec.cmd.Copy_active_to_default = 1 THEN
		gRecCfg.defaultvals.Rec := gRecCfg.active.Rec;
	END_IF;

	IF loc.Rec.cmd.Copy_internal_to_default = 1 THEN
//		Set_Default_Rec;
	END_IF;

	loc.Cfg.status.save_differs_from_active := BOOL_TO_USINT(brsmemcmp(ADR(gRecCfg.save.Cfg),ADR(gRecCfg.active.Cfg), SIZEOF(Global_Cfg_typ)) <> 0);
	loc.Cfg.status.default_differs_from_save := BOOL_TO_USINT(brsmemcmp(ADR(gRecCfg.defaultvals.Cfg),ADR(gRecCfg.save.Cfg), SIZEOF(Global_Cfg_typ)) <> 0);
	loc.Cfg.status.active_differs_from_default := BOOL_TO_USINT(brsmemcmp(ADR(gRecCfg.active.Cfg),ADR(gRecCfg.defaultvals.Cfg), SIZEOF(Global_Cfg_typ)) <> 0);

//	loc.Cfg.status.Invalid := NOT Fcn_Config_Valid(pCfg := ADR(gRecCfg.active.Cfg), pAlarms := ADR(gAlarms));

	loc.Rec.status.save_differs_from_active := BOOL_TO_USINT(brsmemcmp(ADR(gRecCfg.save.Rec),ADR(gRecCfg.active.Rec), SIZEOF(Global_Rec_typ)) <> 0);
	loc.Rec.status.default_differs_from_save := BOOL_TO_USINT(brsmemcmp(ADR(gRecCfg.defaultvals.Rec),ADR(gRecCfg.save.Rec), SIZEOF(Global_Rec_typ)) <> 0);
	loc.Rec.status.active_differs_from_default := BOOL_TO_USINT(brsmemcmp(ADR(gRecCfg.active.Rec),ADR(gRecCfg.defaultvals.Rec), SIZEOF(Global_Rec_typ)) <> 0);

	gAlarms.Unsaved_Recipe_Params := USINT_TO_BOOL(loc.Rec.status.save_differs_from_active);

//	loc.Rec.status.Invalid := NOT Fcn_Recipe_Valid(pRec := ADR(gRecCfg.active.Rec), pAlarms := ADR(gAlarms));

	locCurrentlySelectedRecIsActive := (brsstrcmp(ADR(gRecipe_CSV_UIConnect.Recipe.List.Names[gRecipe_CSV_UIConnect.Recipe.List.SelectedIndex]), ADR(gRecipeName)) = 0);
	locCurrentlySelectedCfgIsActive := (brsstrcmp(ADR(gConfig_CSV_UIConnect.Recipe.List.Names[gConfig_CSV_UIConnect.Recipe.List.SelectedIndex]), ADR(gConfigName)) = 0);

	CASE pRecCfgUIConnect.MessageBox.Type OF
		mpRECIPE_UI_MSG_CONFIRM_LOAD:

		mpRECIPE_UI_MSG_CONFIRM_SAVE:

			IF EDGEPOS(pRecCfgUIConnect.MessageBox.Confirm) THEN
				CASE gHmi.prv.currentPage OF
					HMI_RECIPE_20_SELECT:
						gRecCfg.save.Rec := gRecCfg.active.Rec;
					HMI_CONFIG_30_SELECT:
						gRecCfg.save.Cfg := gRecCfg.active.Cfg;
				END_CASE;
			END_IF;
		mpRECIPE_UI_MSG_CONFIRM_CREATE:

		mpRECIPE_UI_MSG_CONFIRM_DELETE:
			CASE gHmi.prv.currentPage OF
				HMI_RECIPE_20_SELECT:
					IF EDGEPOS(gRecipe_CSV_UIConnect.MessageBox.Confirm) THEN
						IF (brsstrcmp(ADR(gRecipe_CSV_UIConnect.Recipe.List.Names[gRecipe_CSV_UIConnect.Recipe.List.SelectedIndex]), ADR(gRecipeName)) = 0) THEN
							gRecipe_CSV_UIConnect.MessageBox.Confirm := FALSE; //can't delete active recipe
							gRecipe_CSV_UIConnect.MessageBox.Cancel := TRUE;
						END_IF;
					END_IF;
				HMI_CONFIG_30_SELECT:
					IF EDGEPOS(gConfig_CSV_UIConnect.MessageBox.Confirm) THEN
						IF (brsstrcmp(ADR(gConfig_CSV_UIConnect.Recipe.List.Names[gConfig_CSV_UIConnect.Recipe.List.SelectedIndex]), ADR(gConfigName)) = 0) THEN
							gConfig_CSV_UIConnect.MessageBox.Confirm := FALSE; //can't delete active recipe
							gConfig_CSV_UIConnect.MessageBox.Cancel := TRUE;
						END_IF;
					END_IF;
			END_CASE;
	END_CASE;
	//
	IF loc.Rec.HMI.Refresh.DP = 1 THEN
		gRecipe_CSV_UIConnect.Recipe.Refresh := 1;
	END_IF;

	IF loc.Cfg.HMI.Refresh.DP = 1 THEN
		gConfig_CSV_UIConnect.Recipe.Refresh := 1;
	END_IF;

	loc.Rec.HMI.Refresh.DP := 0;
	loc.Rec.HMI.Refresh.Status := DINT_TO_BOOL(gHmiParamTable.selValueFormVisible = 1);
	loc.Rec.HMI.Refresh.Lock := 0;

	loc.Cfg.HMI.Refresh.DP := 0;
	//
	IF loc.Rec.HMI.Save.DP = 1 THEN

		//Make sure listbox selected recipe name is the active one when you are trying to save from a page other than the Rec/Cfg control page (Saving on PVListView page)
		Action_Set_Active_Rec;

		gRecipe_CSV_UIConnect.Recipe.Save := 1;
	END_IF;

	IF loc.Cfg.HMI.Save.DP = 1 THEN
		gConfig_CSV_UIConnect.Recipe.Save := 1;
	END_IF;
	//
	loc.Rec.HMI.Save.DP := 0;
	loc.Rec.HMI.Save.Status := NOT (loc.Rec.status.save_differs_from_active = 1) OR ((NOT (locCurrentlySelectedRecIsActive = 1)) AND gHmi.prv.currentPage = HMI_RECIPE_21_PVLIST) OR DINT_TO_BOOL(gHmiParamTable.selValueFormVisible = 1);
	loc.Rec.HMI.Save.Lock := 0;

	loc.Cfg.HMI.Save.DP := 0;

	//
	IF loc.Rec.HMI.Load.DP = 1 THEN
		gRecipe_CSV_UIConnect.Recipe.Load := 1;
	END_IF;

	IF loc.Cfg.HMI.Load.DP = 1 THEN
		gConfig_CSV_UIConnect.Recipe.Load := 1;
	END_IF;
	//
	loc.Rec.HMI.Load.DP := 0;
	loc.Rec.HMI.Load.Status :=  DINT_TO_BOOL(gHmiParamTable.selValueFormVisible = 1);
	loc.Rec.HMI.Load.Lock := 0;

	loc.Cfg.HMI.Load.DP := 0;
	//
	IF loc.Rec.HMI.Delete.DP = 1 THEN
		gRecipe_CSV_UIConnect.Recipe.Delete := 1;
	END_IF;

	IF loc.Cfg.HMI.Delete.DP = 1 THEN
		gConfig_CSV_UIConnect.Recipe.Delete := 1;
	END_IF;
	//
	loc.Rec.HMI.Delete.DP := 0;
	loc.Rec.HMI.Delete.Status := locCurrentlySelectedRecIsActive OR DINT_TO_BOOL(gHmiParamTable.selValueFormVisible = 1);
	loc.Rec.HMI.Delete.Lock := 0;

	loc.Cfg.HMI.Delete.DP := 0;
	//
	IF loc.Rec.HMI.Overwrite.DP = 1 THEN
		gRecCfg.IO.Rec.I.FileName := gRecipe_CSV_UIConnect.Recipe.List.Names[gRecipe_CSV_UIConnect.Recipe.List.SelectedIndex];
		Recipe_CSV_Control.Save := TRUE;
	END_IF;

	IF loc.Cfg.HMI.Overwrite.DP = 1 THEN
		gRecCfg.IO.Cfg.I.FileName := gConfig_CSV_UIConnect.Recipe.List.Names[gConfig_CSV_UIConnect.Recipe.List.SelectedIndex];
		Config_CSV_Control.Save := TRUE;
	END_IF;
	//
	loc.Rec.HMI.Overwrite.DP := 0;
	//	loc.Rec.HMI.Overwrite.Status := locCurrentlySelectedRecIsActive OR DINT_TO_BOOL(gHmiParamTable.selValueFormVisible = 1);
	loc.Rec.HMI.Overwrite.Status := 1;
	loc.Rec.HMI.Overwrite.Lock := 0;

	IF loc.Rec.HMI.Copy.DP = 1 THEN
		locDTGetTime.enable := 1;
		locDTGetTime();
		locTimeString := '';
		ascDT(locDTGetTime.DT1, ADR(locTimeString), 255);
		gRecCfg.IO.Rec.I.FileName := '';
		gRecCfg.IO.Rec.I.FileName := gRecipeName;
		brsmemset(ADR(gRecCfg.IO.Rec.I.FileName) + brsstrlen(ADR(gRecCfg.IO.Rec.I.FileName)) - 4, 0,1);
		brsstrcat(ADR(gRecCfg.IO.Rec.I.FileName), ADR('_cpy_'));
		brsstrcat(ADR(gRecCfg.IO.Rec.I.FileName), ADR(locTimeString));
		brsstrcat(ADR(gRecCfg.IO.Rec.I.FileName), ADR('.csv'));
		FOR ii_char := 0 TO brsstrlen(ADR(gRecCfg.IO.Rec.I.FileName)) BY 1 DO
			IF brsmemcmp(ADR(gRecCfg.IO.Rec.I.FileName) + ii_char, ADR(':'), 1) = 0 OR brsmemcmp(ADR(gRecCfg.IO.Rec.I.FileName) + ii_char, ADR(' '), 1) = 0 THEN
				brsmemset(ADR(gRecCfg.IO.Rec.I.FileName) + ii_char, 95, 1);
			END_IF;
		END_FOR;
		Recipe_CSV_Control.Save := 1;
	END_IF;

	loc.Rec.HMI.Copy.DP := 0;
	loc.Rec.HMI.Copy.Status := NOT (locCurrentlySelectedRecIsActive = 1) OR DINT_TO_BOOL(gHmiParamTable.selValueFormVisible = 1);
	loc.Rec.HMI.Copy.Lock := 0;

	loc.Cfg.HMI.Refresh.Status := DINT_TO_BOOL(gHmiParamTable.selValueFormVisible = 1);
	loc.Cfg.HMI.Save.Status := DINT_TO_BOOL(gHmiParamTable.selValueFormVisible = 1);
	loc.Cfg.HMI.Load.Status := DINT_TO_BOOL(gHmiParamTable.selValueFormVisible = 1);
	loc.Cfg.HMI.Delete.Status := DINT_TO_BOOL(gHmiParamTable.selValueFormVisible = 1);
	loc.Cfg.HMI.Overwrite.Status := 1;
	loc.Cfg.HMI.Copy.Status := 1;

	locRefreshBeforeCall := gRecipe_CSV_UIConnect.Recipe.Refresh;

	Recipe_CSV_Control;
	Recipe_CSV_RegPar;
	Recipe_CSV_UI;
	pRecCfgUIConnect;
	gRecipe_CSV_UIConnect;

	Config_CSV_Control;
	Config_CSV_RegPar;
	Config_CSV_UI;
	gConfig_CSV_UIConnect;

	IF (NOT gRecipe_CSV_UIConnect.Recipe.Refresh AND locRefreshBeforeCall) OR locFindActiveRecipe = 1 THEN
		bgTimerStart(loc_Timer_Find_Active, Tms(2));
		locFindActiveRecipe := 0;
	END_IF;

//	IF EDGEPOS(bgTimerIsTimeOut(loc_Timer_Find_Active)) THEN
//		FOR ii_recipes := 0 TO 19 BY 1 DO
//			IF (brsstrcmp(ADR(gRecipe_CSV_UIConnect.Recipe.List.Names[ii_recipes]), ADR(gRecipeName)) = 0) THEN
//				gRecipe_CSV_UIConnect.Recipe.List.SelectedIndex := ii_recipes;
//			END_IF;
//		END_FOR;
	//	END_IF;

	IF EDGEPOS(bgTimerIsTimeOut(loc_Timer_Find_Active)) THEN
		Action_Set_Active_Rec;
	END_IF;
	//
	IF Recipe_CSV_Control.CommandDone AND (Recipe_CSV_Control.Save OR Recipe_CSV_Control.Load) THEN
		Recipe_CSV_Control.Save := FALSE;
		Recipe_CSV_Control.Load := FALSE;
		gRecipe_CSV_UIConnect.Recipe.Refresh := 1;
	END_IF;

	IF EDGENEG(gRecipe_CSV_UIConnect.Status = mpRECIPE_UI_STATUS_SAVE) THEN
//		gRecipeName := Recipe_CSV_Control.Info.LastLoadedRecipe;
		gRecCfg.save.Rec := gRecCfg.active.Rec;
	END_IF;

	IF EDGENEG(gRecipe_CSV_UIConnect.Status = mpRECIPE_UI_STATUS_LOAD) THEN
		gRecCfg.IO.Rec.O.Initial_Load := 1;
		gRecipeName := Recipe_CSV_Control.Info.LastLoadedRecipe;
		gRecCfg.active.Rec := gRecCfg.save.Rec;
	END_IF;

	loc.Rec.cmd.Copy_default_to_save := FALSE;
	loc.Rec.cmd.Copy_default_to_active := FALSE;
	loc.Rec.cmd.Copy_save_to_active := FALSE;
	loc.Rec.cmd.Copy_save_to_default := FALSE;
	loc.Rec.cmd.Copy_active_to_save := FALSE;
	loc.Rec.cmd.Copy_active_to_default := FALSE;
	loc.Rec.cmd.Copy_internal_to_default := FALSE;

	bgTimerCyclic(loc_Timer_Find_Active);
	//

	IF Config_CSV_Control.CommandDone AND (Config_CSV_Control.Save OR Config_CSV_Control.Load) THEN
		Config_CSV_Control.Save := FALSE;
		Config_CSV_Control.Load := FALSE;
		gConfig_CSV_UIConnect.Recipe.Refresh := 1;
	END_IF;

	IF EDGENEG(gConfig_CSV_UIConnect.Status = mpRECIPE_UI_STATUS_SAVE) THEN
//		gConfigName := Config_CSV_Control.Info.LastLoadedRecipe;
		gRecCfg.save.Cfg := gRecCfg.active.Cfg;
	END_IF;

	IF EDGENEG(gConfig_CSV_UIConnect.Status = mpRECIPE_UI_STATUS_LOAD) THEN
		gConfigName := Config_CSV_Control.Info.LastLoadedRecipe;
		gRecCfg.active.Cfg := gRecCfg.save.Cfg;
	END_IF;

	loc.Cfg.cmd.Copy_default_to_save := FALSE;
	loc.Cfg.cmd.Copy_default_to_active := FALSE;
	loc.Cfg.cmd.Copy_save_to_active := FALSE;
	loc.Cfg.cmd.Copy_save_to_default := FALSE;
	loc.Cfg.cmd.Copy_active_to_save := FALSE;
	loc.Cfg.cmd.Copy_active_to_default := FALSE;
	loc.Cfg.cmd.Copy_internal_to_default := FALSE;
	//
END_PROGRAM
```

#### Init.st
```iecst
PROGRAM _INIT
	IF gRecCfg.active.Cfg.MagicPrefix <> DEFINE_CONSTANT_MAGIC_PREFIX OR gRecCfg.save.Cfg.MagicPrefix <> DEFINE_CONSTANT_MAGIC_PREFIX OR gRecCfg.defaultvals.Cfg.MagicPrefix <> DEFINE_CONSTANT_MAGIC_PREFIX
		OR gRecCfg.active.Cfg.MagicSuffix <> DEFINE_CONSTANT_MAGIC_SUFFIX OR gRecCfg.save.Cfg.MagicSuffix <> DEFINE_CONSTANT_MAGIC_SUFFIX OR gRecCfg.defaultvals.Cfg.MagicSuffix <> DEFINE_CONSTANT_MAGIC_SUFFIX
		OR gRecCfg.active.Rec.MagicPrefix <> DEFINE_CONSTANT_MAGIC_PREFIX OR gRecCfg.save.Rec.MagicPrefix <> DEFINE_CONSTANT_MAGIC_PREFIX OR gRecCfg.defaultvals.Rec.MagicPrefix <> DEFINE_CONSTANT_MAGIC_PREFIX
		OR gRecCfg.active.Rec.MagicSuffix <> DEFINE_CONSTANT_MAGIC_SUFFIX OR gRecCfg.save.Rec.MagicSuffix <> DEFINE_CONSTANT_MAGIC_SUFFIX OR gRecCfg.defaultvals.Rec.MagicSuffix <> DEFINE_CONSTANT_MAGIC_SUFFIX
		THEN

		brsmemset(ADR(gRecCfg.defaultvals.Cfg), 0, SIZEOF(Global_Cfg_typ));
		brsmemset(ADR(gRecCfg.save.Cfg), 0, SIZEOF(Global_Cfg_typ));
		brsmemset(ADR(gRecCfg.active.Cfg), 0, SIZEOF(Global_Cfg_typ));

		brsmemset(ADR(gRecCfg.defaultvals.Rec), 0, SIZEOF(Global_Rec_typ));
		brsmemset(ADR(gRecCfg.save.Rec), 0, SIZEOF(Global_Rec_typ));
		brsmemset(ADR(gRecCfg.active.Rec), 0, SIZEOF(Global_Rec_typ));

		brsmemset(ADR(gStatistics), 0, SIZEOF(AS3500HS_Stats_typ));

		gRecCfg.active.Cfg.MagicPrefix := DEFINE_CONSTANT_MAGIC_PREFIX;
		gRecCfg.save.Cfg.MagicPrefix:= DEFINE_CONSTANT_MAGIC_PREFIX;
		gRecCfg.defaultvals.Cfg.MagicPrefix:= DEFINE_CONSTANT_MAGIC_PREFIX;

		gRecCfg.active.Cfg.MagicSuffix := DEFINE_CONSTANT_MAGIC_SUFFIX;
		gRecCfg.save.Cfg.MagicSuffix:= DEFINE_CONSTANT_MAGIC_SUFFIX;
		gRecCfg.defaultvals.Cfg.MagicSuffix:= DEFINE_CONSTANT_MAGIC_SUFFIX;

		gRecCfg.active.Rec.MagicPrefix := DEFINE_CONSTANT_MAGIC_PREFIX;
		gRecCfg.save.Rec.MagicPrefix:= DEFINE_CONSTANT_MAGIC_PREFIX;
		gRecCfg.defaultvals.Rec.MagicPrefix:= DEFINE_CONSTANT_MAGIC_PREFIX;

		gRecCfg.active.Rec.MagicSuffix := DEFINE_CONSTANT_MAGIC_SUFFIX;
		gRecCfg.save.Rec.MagicSuffix:= DEFINE_CONSTANT_MAGIC_SUFFIX;
		gRecCfg.defaultvals.Rec.MagicSuffix:= DEFINE_CONSTANT_MAGIC_SUFFIX;

		Set_Default_Config_Values(pCfg := ADR(gRecCfg.defaultvals.Cfg));
		Set_Default_Config_Values(pCfg := ADR(gRecCfg.save.Cfg));
		Set_Default_Config_Values(pCfg := ADR(gRecCfg.active.Cfg));

		gConfigName := 'No Config';

		Set_Default_Recipe_Values(pRec := ADR(gRecCfg.defaultvals.Rec));
		Set_Default_Recipe_Values(pRec := ADR(gRecCfg.save.Rec));
		Set_Default_Recipe_Values(pRec := ADR(gRecCfg.active.Rec));

		gRecipeName := 'No Recipe';

//		gAlarms.RecCfg.Default_Rec_Set := TRUE;

//		gAlarms.RecCfg.Default_Cfg_Set := TRUE;

//		SYSreset(1, 1);
	END_IF;

	gRecCfg.IO.Rec.I.FileName := 'rec1';
	gRecCfg.IO.Cfg.I.FileName := 'cfg1';

	Recipe_CSV_Control.MpLink := ADR(Recipe_CSV_MpLink);
	Recipe_CSV_Control.Enable := TRUE;
	Recipe_CSV_Control.DeviceName := ADR('Recipe');
	Recipe_CSV_Control.FileName := ADR(gRecCfg.IO.Rec.I.FileName);
	Recipe_CSV_Control.Category := ADR('Recipe');
	Recipe_CSV_Control.Header := ADR(Recipe_CSV_Header);

	Config_CSV_Control.MpLink := ADR(Config_CSV_MpLink);
	Config_CSV_Control.Enable := TRUE;
	Config_CSV_Control.DeviceName := ADR('Config');
	Config_CSV_Control.FileName := ADR(gRecCfg.IO.Cfg.I.FileName);
	Config_CSV_Control.Category := ADR('Config');
	Config_CSV_Control.Header := ADR(Config_CSV_Header);

	Recipe_CSV_RegPar.MpLink := ADR(Recipe_CSV_MpLink);
	Recipe_CSV_RegPar.Enable := TRUE;
	Recipe_CSV_RegPar.PVName := ADR('gRecCfg.save.Rec');
	Recipe_CSV_RegPar.Category := ADR('Recipe');

	Config_CSV_RegPar.MpLink := ADR(Config_CSV_MpLink);
	Config_CSV_RegPar.Enable := TRUE;
	Config_CSV_RegPar.PVName := ADR('gRecCfg.save.Cfg');
	Config_CSV_RegPar.Category := ADR('Config');

	Recipe_CSV_UI.MpLink := ADR(Recipe_CSV_MpLink);
	Recipe_CSV_UI.Enable := TRUE;
	Recipe_CSV_UI.UIConnect := ADR(gRecipe_CSV_UIConnect);

	Config_CSV_UI.MpLink := ADR(Config_CSV_MpLink);
	Config_CSV_UI.Enable := TRUE;
	Config_CSV_UI.UIConnect := ADR(gConfig_CSV_UIConnect);

	Recipe_CSV_UI.UISetup.RecipeListSize := 20;
	Recipe_CSV_UI.UISetup.RecipeListScrollWindow := 1;
	Recipe_CSV_UI.UISetup.Confirmation.RecipeCreate := TRUE;
	Recipe_CSV_UI.UISetup.Confirmation.RecipeLoad := TRUE;
	Recipe_CSV_UI.UISetup.Confirmation.RecipeSave := TRUE;
	Recipe_CSV_UI.UISetup.Confirmation.RecipeDelete := TRUE;

	Config_CSV_UI.UISetup.RecipeListSize := 20;
	Config_CSV_UI.UISetup.RecipeListScrollWindow := 1;
	Config_CSV_UI.UISetup.Confirmation.RecipeCreate := TRUE;
	Config_CSV_UI.UISetup.Confirmation.RecipeLoad := TRUE;
	Config_CSV_UI.UISetup.Confirmation.RecipeSave := TRUE;
	Config_CSV_UI.UISetup.Confirmation.RecipeDelete := TRUE;

	pRecCfgUIConnect ACCESS ADR(gRecipe_CSV_UIConnect);
	pCmd ACCESS ADR(loc.Rec.HMI);

	gRecipe_CSV_UIConnect.New.FileName := 'Rec_Name';
	gConfig_CSV_UIConnect.New.FileName := 'Cfg_Name';

	Recipe_CSV_Control;
	Recipe_CSV_RegPar;
	Recipe_CSV_UI;

	Config_CSV_Control;
	Config_CSV_RegPar;
	Config_CSV_UI;

	Alarm_Recipe_UI.MpLink := ADR(Recipe_CSV_MpLink);
	Alarm_Recipe_UI.Enable := TRUE;
	Alarm_Recipe_UI.Mode := mpALARM_BASIC_UI_MODE_ALL;

	Alarm_Recipe_UI.UISetup.ImageSize := 20;
	Alarm_Recipe_UI.UISetup.AlarmImage := ADR(Alarm_Recipe.AlarmImage[0]);
	Alarm_Recipe_UI.UISetup.AcknowledgeImage := ADR(Alarm_Recipe.AcknowledgeImage[0]);
	Alarm_Recipe_UI.UISetup.AddInfoStringSize := 100;
	Alarm_Recipe_UI.UISetup.AddInfo := ADR(Alarm_Recipe.AddInfo[0]);

	Alarm_Recipe;
	Alarm_Recipe_UI();

	Alarm_Config_UI.MpLink := ADR(Config_CSV_MpLink);
	Alarm_Config_UI.Enable := TRUE;
	Alarm_Config_UI.Mode := mpALARM_BASIC_UI_MODE_ALL;

	Alarm_Config_UI.UISetup.ImageSize := 20;
	Alarm_Config_UI.UISetup.AlarmImage := ADR(Alarm_Config.AlarmImage[0]);
	Alarm_Config_UI.UISetup.AcknowledgeImage := ADR(Alarm_Config.AcknowledgeImage[0]);
	Alarm_Config_UI.UISetup.AddInfoStringSize := 100;
	Alarm_Config_UI.UISetup.AddInfo := ADR(Alarm_Config.AddInfo[0]);

	Alarm_Config;
	Alarm_Config_UI();
END_PROGRAM
```

#### Set_Default_Config_Values.st
```iecst
FUNCTION Set_Default_Config_Values

	pCfg.HMI.passwordSetup := '1111';
	pCfg.HMI.passwordEngineer := '2222';
	pCfg.HMI.passwordFactory := '3333';

	pCfg.Control.N_Encoder_Bits_SingleTurn := 12;
	pCfg.Control.Encoder_Position_Home := 0;

	pCfg.Control.Debounce_PiP.Timer_On := 0.02;
	pCfg.Control.Debounce_PiP.Timer_Off := 0.02;

	pCfg.Control.Threshold_AccelDecel_Trans_RPM := 0.05;
	pCfg.Control.T_Exit_Decel_Automatically := 9999;
	pCfg.Control.Target_Present_Pulse_Time_S := 0.05;

	pCfg.Control.Sim_Encoder := 0;
	pCfg.Control.Sim_Encoder_Cycles := 1;
	pCfg.Control.Sim_Encoder_Counts := 2;

	pCfg.Dispense[0].Disable := FALSE;
	pCfg.Dispense[1].Disable := FALSE;

	Set_Default_Config_Values := 0;
END_FUNCTION
```

#### Set_Default_Recipe_Values.st
```iecst
FUNCTION Set_Default_Recipe_Values

	pRec.Control.N_Targets_On_Dial := 18;

	FOR ii_dispense_units := 0 TO MAX_IDX_VALVES BY 1 DO
		pRec.Dispense[ii_dispense_units].Enable := 0;
		pRec.Dispense[ii_dispense_units].Disp_Valve_Edgemode_Pulse_TO_ms := 25;
		pRec.Dispense[ii_dispense_units].Extra_Shots_Per_VBlock := 0;
		pRec.Dispense[ii_dispense_units].Time_Offset_Additional_Shots := 0.1;
		pRec.Dispense[ii_dispense_units].Target_Offset := 3 + 2*ii_dispense_units;
	END_FOR;

	Set_Default_Recipe_Values := 0;
END_FUNCTION
```
